Universal Robots URScript: draw_back.script

def unnamed():
  set_tcp(p[0.0,0.0,0.0,0.0,0.0,0.0])
  set_safety_mode_transition_hardness(1)
  set_tool_communication(True, 1000000, 2, 1, 1.5, 3.5)
  set_tool_output_mode(0)
  set_tool_digital_output_mode(0, 1)
  set_tool_digital_output_mode(1, 1)
  set_tool_voltage(0)
  step_count_92a71080_320b_48c3_b710_fb27a0ae3266 = 0.0
  thread Step_Counter_Thread_29a6b4c0_57cd_4359_a365_f92f2370702e():
    while (True):
      step_count_92a71080_320b_48c3_b710_fb27a0ae3266 = step_count_92a71080_320b_48c3_b710_fb27a0ae3266 + 1.0
      sync()
    end
  end
  run Step_Counter_Thread_29a6b4c0_57cd_4359_a365_f92f2370702e()
  set_gravity([0.0, 0.0, 9.82])
  set_standard_analog_input_domain(0, 1)
  set_standard_analog_input_domain(1, 1)
  set_tool_analog_input_domain(0, 1)
  set_tool_analog_input_domain(1, 1)
  set_analog_outputdomain(0, 0)
  set_analog_outputdomain(1, 0)
  set_input_actions_to_default()
  set_target_payload(1.070000, [0.002000, 0.003000, 0.057000], [0.001723, 0.001723, 0.001723, 0.000000, 0.000000, 0.000000])
  global Plane_1=p[-0.700006141123905,1.3454883874109249E-6,0.3910559577028425,-1.2089868272251132,-1.2089999932245832,1.20858562628424]
  global Plane_2=p[0.0,0.0,0.0,0.0,0.0,0.0]
  global Point_1=p[0.6913645118948067,-0.12399382748223003,0.49223711947071,-1.2983729986843258,1.1259514972191385,-1.2203503861141718]
  $ 1 "Robot Program"
  $ 2 "Script: draw_back.script"
  def Machining1():
    # Default parameters:
    global speed_ms = 0.3
    global speed_rads = 0.75
    global accel_mss = 3
    global accel_radss = 1.2
    global blend_radius_m = 0.001

    # Add subprograms here
    # Start of main program
    # Program generated by RoboDK v5.6.5 for UR10e on 18/10/2023 16:38:27
    # Using nominal kinematics.
    blend_radius_m = 0.001
    speed_ms = 1.000
    # set_reference(p[0.335000, -0.152000, 0.000000, 0.000000, 0.000000, 0.000000])
    set_tcp(p[0.000000, 0.000000, 0.252000, 0.000000, 0.000000, 0.000000])
    # Show Tool
    movej([0.136763, -1.127639, -2.609664, -0.975086, 1.570796, 1.707559],accel_radss,speed_rads,0,blend_radius_m)
    movel([0.136763, -1.187625, -2.647719, -0.877045, 1.570796, 1.707559],accel_mss,speed_ms,0,blend_radius_m)
    speed_ms = 1.000
    movel([0.136763, -1.198811, -2.653791, -0.859786, 1.570796, 1.707559],accel_mss,speed_ms,0,blend_radius_m)
    movel([0.136763, -1.222268, -2.665681, -0.824440, 1.570796, 1.707559],accel_mss,speed_ms,0,blend_radius_m)
    movel([0.124896, -1.226310, -2.663645, -0.822433, 1.570796, 1.695693],accel_mss,speed_ms,0,blend_radius_m)
    movel([0.124896, -1.202890, -2.651801, -0.857697, 1.570796, 1.695693],accel_mss,speed_ms,0,blend_radius_m)
    movel([0.135681, -1.206174, -2.650186, -0.856029, 1.570796, 1.706478],accel_mss,speed_ms,0,blend_radius_m)
    movel([0.135681, -1.229564, -2.661993, -0.820832, 1.570796, 1.706478],accel_mss,speed_ms,0,blend_radius_m)
    movel([0.123913, -1.233531, -2.659963, -0.818895, 1.570796, 1.694709],accel_mss,speed_ms,0,blend_radius_m)
    movel([0.123913, -1.210179, -2.648200, -0.854011, 1.570796, 1.694709],accel_mss,speed_ms,0,blend_radius_m)
    movel([0.131108, -1.200743, -2.652851, -0.858795, 1.570796, 1.701904],accel_mss,speed_ms,0,blend_radius_m)
    movel([0.131108, -1.224182, -2.664719, -0.823487, 1.570796, 1.701904],accel_mss,speed_ms,0,blend_radius_m)
    movel([0.130073, -1.231443, -2.661034, -0.819912, 1.570796, 1.700869],accel_mss,speed_ms,0,blend_radius_m)
    movel([0.130073, -1.208071, -2.649247, -0.855071, 1.570796, 1.700869],accel_mss,speed_ms,0,blend_radius_m)
    movel([0.135147, -1.209825, -2.648376, -0.854188, 1.570796, 1.705943],accel_mss,speed_ms,0,blend_radius_m)
    movel([0.135147, -1.233181, -2.660143, -0.819066, 1.570796, 1.705943],accel_mss,speed_ms,0,blend_radius_m)
    movel([0.134512, -1.233881, -2.659782, -0.818725, 1.570796, 1.705309],accel_mss,speed_ms,0,blend_radius_m)
    movel([0.134995, -1.234210, -2.659613, -0.818566, 1.570796, 1.705792],accel_mss,speed_ms,0,blend_radius_m)
    movel([0.135630, -1.233511, -2.659973, -0.818905, 1.570796, 1.706426],accel_mss,speed_ms,0,blend_radius_m)
    movel([0.135147, -1.233181, -2.660143, -0.819066, 1.570796, 1.705943],accel_mss,speed_ms,0,blend_radius_m)
    movel([0.135147, -1.209825, -2.648376, -0.854188, 1.570796, 1.705943],accel_mss,speed_ms,0,blend_radius_m)
    movel([0.131163, -1.211657, -2.647462, -0.853270, 1.570796, 1.701959],accel_mss,speed_ms,0,blend_radius_m)
    movel([0.131163, -1.234995, -2.659208, -0.818185, 1.570796, 1.701959],accel_mss,speed_ms,0,blend_radius_m)
    movel([0.123358, -1.237621, -2.657850, -0.816918, 1.570796, 1.694154],accel_mss,speed_ms,0,blend_radius_m)
    movel([0.123358, -1.214308, -2.646133, -0.851948, 1.570796, 1.694154],accel_mss,speed_ms,0,blend_radius_m)
    movel([0.118731, -1.205544, -2.650497, -0.856348, 1.570796, 1.689527],accel_mss,speed_ms,0,blend_radius_m)
    movel([0.118731, -1.228940, -2.662311, -0.821138, 1.570796, 1.689527],accel_mss,speed_ms,0,blend_radius_m)
    movel([0.109176, -1.232299, -2.660595, -0.819495, 1.570796, 1.679972],accel_mss,speed_ms,0,blend_radius_m)
    movel([0.107432, -1.233406, -2.660027, -0.818956, 1.570796, 1.678228],accel_mss,speed_ms,0,blend_radius_m)
    movel([0.106751, -1.234624, -2.659400, -0.818365, 1.570796, 1.677547],accel_mss,speed_ms,0,blend_radius_m)
    movel([0.106631, -1.235641, -2.658875, -0.817873, 1.570796, 1.677427],accel_mss,speed_ms,0,blend_radius_m)
    movel([0.106631, -1.212309, -2.647136, -0.852944, 1.570796, 1.677427],accel_mss,speed_ms,0,blend_radius_m)
    movel([0.114988, -1.205377, -2.650579, -0.856433, 1.570796, 1.685784],accel_mss,speed_ms,0,blend_radius_m)
    movel([0.114988, -1.228774, -2.662396, -0.821219, 1.570796, 1.685784],accel_mss,speed_ms,0,blend_radius_m)
    movel([0.114535, -1.232368, -2.660560, -0.819461, 1.570796, 1.685331],accel_mss,speed_ms,0,blend_radius_m)
    movel([0.114535, -1.209004, -2.648784, -0.854601, 1.570796, 1.685331],accel_mss,speed_ms,0,blend_radius_m)
    movel([0.117997, -1.211242, -2.647669, -0.853477, 1.570796, 1.688794],accel_mss,speed_ms,0,blend_radius_m)
    movel([0.117997, -1.234584, -2.659420, -0.818384, 1.570796, 1.688794],accel_mss,speed_ms,0,blend_radius_m)
    movel([0.106273, -1.238681, -2.657299, -0.816409, 1.570796, 1.677069],accel_mss,speed_ms,0,blend_radius_m)
    movel([0.106273, -1.215379, -2.645594, -0.851416, 1.570796, 1.677069],accel_mss,speed_ms,0,blend_radius_m)
    movel([0.111851, -1.213399, -2.646590, -0.852400, 1.570796, 1.682647],accel_mss,speed_ms,0,blend_radius_m)
    movel([0.111851, -1.236721, -2.658316, -0.817352, 1.570796, 1.682647],accel_mss,speed_ms,0,blend_radius_m)
    movel([0.113335, -1.237661, -2.657829, -0.816899, 1.570796, 1.684132],accel_mss,speed_ms,0,blend_radius_m)
    movel([0.113766, -1.238482, -2.657402, -0.816505, 1.570796, 1.684562],accel_mss,speed_ms,0,blend_radius_m)
    movel([0.113575, -1.240002, -2.656611, -0.815777, 1.570796, 1.684371],accel_mss,speed_ms,0,blend_radius_m)
    movel([0.112893, -1.241205, -2.655982, -0.815202, 1.570796, 1.683689],accel_mss,speed_ms,0,blend_radius_m)
    movel([0.111165, -1.242286, -2.655416, -0.814687, 1.570796, 1.681962],accel_mss,speed_ms,0,blend_radius_m)
    movel([0.105623, -1.244218, -2.654400, -0.813771, 1.570796, 1.676419],accel_mss,speed_ms,0,blend_radius_m)
    movel([0.105623, -1.220971, -2.642758, -0.848660, 1.570796, 1.676419],accel_mss,speed_ms,0,blend_radius_m)
    movel([0.112197, -1.227862, -2.639215, -0.845312, 1.570796, 1.682993],accel_mss,speed_ms,0,blend_radius_m)
    movel([0.112197, -1.251037, -2.650780, -0.810572, 1.570796, 1.682993],accel_mss,speed_ms,0,blend_radius_m)
    movel([0.104520, -1.253671, -2.649367, -0.809351, 1.570796, 1.675316],accel_mss,speed_ms,0,blend_radius_m)
    movel([0.104520, -1.230524, -2.637832, -0.844033, 1.570796, 1.675316],accel_mss,speed_ms,0,blend_radius_m)
    movel([0.110550, -1.228429, -2.638921, -0.845039, 1.570796, 1.681347],accel_mss,speed_ms,0,blend_radius_m)
    movel([0.110550, -1.251599, -2.650480, -0.810311, 1.570796, 1.681347],accel_mss,speed_ms,0,blend_radius_m)
    movel([0.111771, -1.250229, -2.651212, -0.810948, 1.570796, 1.682568],accel_mss,speed_ms,0,blend_radius_m)
    movel([0.112445, -1.249045, -2.651844, -0.811501, 1.570796, 1.683241],accel_mss,speed_ms,0,blend_radius_m)
    movel([0.112632, -1.247546, -2.652640, -0.812202, 1.570796, 1.683428],accel_mss,speed_ms,0,blend_radius_m)
    movel([0.112205, -1.246735, -2.653071, -0.812584, 1.570796, 1.683001],accel_mss,speed_ms,0,blend_radius_m)
    movel([0.111225, -1.246113, -2.653400, -0.812876, 1.570796, 1.682021],accel_mss,speed_ms,0,blend_radius_m)
    movel([0.109629, -1.246184, -2.653362, -0.812843, 1.570796, 1.680426],accel_mss,speed_ms,0,blend_radius_m)
    movel([0.108525, -1.246566, -2.653160, -0.812663, 1.570796, 1.679321],accel_mss,speed_ms,0,blend_radius_m)
    movel([0.106810, -1.247640, -2.652591, -0.812159, 1.570796, 1.677606],accel_mss,speed_ms,0,blend_radius_m)
    movel([0.105590, -1.249019, -2.651857, -0.811513, 1.570796, 1.676386],accel_mss,speed_ms,0,blend_radius_m)
    movel([0.104923, -1.250204, -2.651225, -0.810959, 1.570796, 1.675720],accel_mss,speed_ms,0,blend_radius_m)
    movel([0.104750, -1.251692, -2.650430, -0.810267, 1.570796, 1.675546],accel_mss,speed_ms,0,blend_radius_m)
    movel([0.105183, -1.252493, -2.650000, -0.809896, 1.570796, 1.675979],accel_mss,speed_ms,0,blend_radius_m)
    movel([0.106163, -1.253104, -2.649672, -0.809613, 1.570796, 1.676960],accel_mss,speed_ms,0,blend_radius_m)
    movel([0.106163, -1.229951, -2.638130, -0.844308, 1.570796, 1.676960],accel_mss,speed_ms,0,blend_radius_m)
    movel([0.111704, -1.231871, -2.637129, -0.843390, 1.570796, 1.682501],accel_mss,speed_ms,0,blend_radius_m)
    movel([0.111704, -1.255003, -2.648649, -0.808736, 1.570796, 1.682501],accel_mss,speed_ms,0,blend_radius_m)
    movel([0.104062, -1.257611, -2.647238, -0.807540, 1.570796, 1.674858],accel_mss,speed_ms,0,blend_radius_m)
    movel([0.104062, -1.234506, -2.635747, -0.842136, 1.570796, 1.674858],accel_mss,speed_ms,0,blend_radius_m)
    movel([0.109519, -1.232620, -2.636737, -0.843032, 1.570796, 1.680315],accel_mss,speed_ms,0,blend_radius_m)
    movel([0.109519, -1.255745, -2.648249, -0.808395, 1.570796, 1.680315],accel_mss,speed_ms,0,blend_radius_m)
    movel([0.110975, -1.256669, -2.647749, -0.807971, 1.570796, 1.681772],accel_mss,speed_ms,0,blend_radius_m)
    movel([0.111399, -1.257470, -2.647314, -0.807605, 1.570796, 1.682195],accel_mss,speed_ms,0,blend_radius_m)
    movel([0.111216, -1.258945, -2.646512, -0.806931, 1.570796, 1.682013],accel_mss,speed_ms,0,blend_radius_m)
    movel([0.110551, -1.260110, -2.645877, -0.806401, 1.570796, 1.681348],accel_mss,speed_ms,0,blend_radius_m)
    movel([0.108863, -1.261149, -2.645310, -0.805930, 1.570796, 1.679659],accel_mss,speed_ms,0,blend_radius_m)
    movel([0.103439, -1.262988, -2.644301, -0.805100, 1.570796, 1.674236],accel_mss,speed_ms,0,blend_radius_m)
    movel([0.103439, -1.239944, -2.632871, -0.839574, 1.570796, 1.674236],accel_mss,speed_ms,0,blend_radius_m)
    movel([0.114338, -1.240023, -2.632829, -0.839537, 1.570796, 1.685135],accel_mss,speed_ms,0,blend_radius_m)
    movel([0.114338, -1.263067, -2.644258, -0.805064, 1.570796, 1.685135],accel_mss,speed_ms,0,blend_radius_m)
    movel([0.102991, -1.266871, -2.642159, -0.803359, 1.570796, 1.673788],accel_mss,speed_ms,0,blend_radius_m)
    movel([0.102991, -1.243871, -2.630773, -0.837745, 1.570796, 1.673788],accel_mss,speed_ms,0,blend_radius_m)
    movel([0.109955, -1.246207, -2.629516, -0.836666, 1.570796, 1.680751],accel_mss,speed_ms,0,blend_radius_m)
    movel([0.109955, -1.269180, -2.640876, -0.802333, 1.570796, 1.680751],accel_mss,speed_ms,0,blend_radius_m)
    movel([0.105150, -1.266141, -2.642563, -0.803685, 1.570796, 1.675946],accel_mss,speed_ms,0,blend_radius_m)
    movel([0.105150, -1.243132, -2.631169, -0.838088, 1.570796, 1.675946],accel_mss,speed_ms,0,blend_radius_m)
    movel([0.107078, -1.244359, -2.630511, -0.837519, 1.570796, 1.677874],accel_mss,speed_ms,0,blend_radius_m)
    movel([0.107078, -1.267353, -2.641891, -0.803144, 1.570796, 1.677874],accel_mss,speed_ms,0,blend_radius_m)
    movel([0.102382, -1.272173, -2.639204, -0.801013, 1.570796, 1.673178],accel_mss,speed_ms,0,blend_radius_m)
    movel([0.102382, -1.249235, -2.627877, -0.835277, 1.570796, 1.673178],accel_mss,speed_ms,0,blend_radius_m)
    movel([0.108723, -1.256402, -2.623955, -0.832032, 1.570796, 1.679519],accel_mss,speed_ms,0,blend_radius_m)
    movel([0.108723, -1.279255, -2.635202, -0.797933, 1.570796, 1.679519],accel_mss,speed_ms,0,blend_radius_m)
    movel([0.100970, -1.284533, -2.632178, -0.795678, 1.570796, 1.671766],accel_mss,speed_ms,0,blend_radius_m)
    movel([0.100970, -1.261746, -2.620991, -0.829652, 1.570796, 1.671766],accel_mss,speed_ms,0,blend_radius_m)
    movel([0.108032, -1.262159, -2.620760, -0.829470, 1.570796, 1.678828],accel_mss,speed_ms,0,blend_radius_m)
    movel([0.108032, -1.284942, -2.631943, -0.795505, 1.570796, 1.678828],accel_mss,speed_ms,0,blend_radius_m)
    movel([0.100970, -1.284533, -2.632178, -0.795678, 1.570796, 1.671766],accel_mss,speed_ms,0,blend_radius_m)
    movel([0.098961, -1.284292, -2.632317, -0.795780, 1.570796, 1.669758],accel_mss,speed_ms,0,blend_radius_m)
    movel([0.098008, -1.283703, -2.632656, -0.796030, 1.570796, 1.668804],accel_mss,speed_ms,0,blend_radius_m)
    movel([0.097582, -1.282937, -2.633096, -0.796356, 1.570796, 1.668379],accel_mss,speed_ms,0,blend_radius_m)
    movel([0.097634, -1.282466, -2.633367, -0.796557, 1.570796, 1.668431],accel_mss,speed_ms,0,blend_radius_m)
    movel([0.097634, -1.259652, -2.622156, -0.830581, 1.570796, 1.668431],accel_mss,speed_ms,0,blend_radius_m)
    movel([0.107462, -1.266919, -2.618088, -0.827381, 1.570796, 1.678259],accel_mss,speed_ms,0,blend_radius_m)
    movel([0.107462, -1.289643, -2.629218, -0.793529, 1.570796, 1.678259],accel_mss,speed_ms,0,blend_radius_m)
    movel([0.107050, -1.288875, -2.629665, -0.793849, 1.570796, 1.677846],accel_mss,speed_ms,0,blend_radius_m)
    movel([0.106111, -1.288277, -2.630012, -0.794100, 1.570796, 1.676908],accel_mss,speed_ms,0,blend_radius_m)
    movel([0.104589, -1.288319, -2.629988, -0.794082, 1.570796, 1.675386],accel_mss,speed_ms,0,blend_radius_m)
    movel([0.103537, -1.288662, -2.629789, -0.793939, 1.570796, 1.674334],accel_mss,speed_ms,0,blend_radius_m)
    movel([0.101907, -1.289644, -2.629217, -0.793528, 1.570796, 1.672703],accel_mss,speed_ms,0,blend_radius_m)
    movel([0.100750, -1.290921, -2.628472, -0.792996, 1.570796, 1.671547],accel_mss,speed_ms,0,blend_radius_m)
    movel([0.100120, -1.292024, -2.627826, -0.792538, 1.570796, 1.670917],accel_mss,speed_ms,0,blend_radius_m)
    movel([0.099963, -1.293419, -2.627008, -0.791962, 1.570796, 1.670759],accel_mss,speed_ms,0,blend_radius_m)
    movel([0.100380, -1.294178, -2.626562, -0.791649, 1.570796, 1.671177],accel_mss,speed_ms,0,blend_radius_m)
    movel([0.101319, -1.294766, -2.626216, -0.791407, 1.570796, 1.672116],accel_mss,speed_ms,0,blend_radius_m)
    movel([0.102832, -1.294723, -2.626241, -0.791425, 1.570796, 1.673628],accel_mss,speed_ms,0,blend_radius_m)
    movel([0.103877, -1.294386, -2.626440, -0.791563, 1.570796, 1.674673],accel_mss,speed_ms,0,blend_radius_m)
    movel([0.105499, -1.293417, -2.627010, -0.791963, 1.570796, 1.676295],accel_mss,speed_ms,0,blend_radius_m)
    movel([0.106656, -1.292149, -2.627754, -0.792487, 1.570796, 1.677453],accel_mss,speed_ms,0,blend_radius_m)
    movel([0.107293, -1.291046, -2.628399, -0.792944, 1.570796, 1.678089],accel_mss,speed_ms,0,blend_radius_m)
    movel([0.107462, -1.289643, -2.629218, -0.793529, 1.570796, 1.678259],accel_mss,speed_ms,0,blend_radius_m)
    movel([0.107462, -1.266919, -2.618088, -0.827381, 1.570796, 1.678259],accel_mss,speed_ms,0,blend_radius_m)
    movel([0.106620, -1.273998, -2.614064, -0.824327, 1.570796, 1.677416],accel_mss,speed_ms,0,blend_radius_m)
    movel([0.106620, -1.296631, -2.625115, -0.790643, 1.570796, 1.677416],accel_mss,speed_ms,0,blend_radius_m)
    movel([0.101416, -1.298298, -2.624127, -0.789964, 1.570796, 1.672213],accel_mss,speed_ms,0,blend_radius_m)
    movel([0.099805, -1.299262, -2.623554, -0.789573, 1.570796, 1.670601],accel_mss,speed_ms,0,blend_radius_m)
    movel([0.099182, -1.300349, -2.622906, -0.789134, 1.570796, 1.669978],accel_mss,speed_ms,0,blend_radius_m)
    movel([0.099027, -1.301727, -2.622084, -0.788579, 1.570796, 1.669824],accel_mss,speed_ms,0,blend_radius_m)
    movel([0.099442, -1.302476, -2.621635, -0.788278, 1.570796, 1.670239],accel_mss,speed_ms,0,blend_radius_m)
    movel([0.100838, -1.303353, -2.621109, -0.787927, 1.570796, 1.671634],accel_mss,speed_ms,0,blend_radius_m)
    movel([0.100838, -1.280809, -2.610134, -0.821446, 1.570796, 1.671634],accel_mss,speed_ms,0,blend_radius_m)
    movel([0.106010, -1.279142, -2.611101, -0.822146, 1.570796, 1.676806],accel_mss,speed_ms,0,blend_radius_m)
    movel([0.106010, -1.301708, -2.622095, -0.788586, 1.570796, 1.676806],accel_mss,speed_ms,0,blend_radius_m)
    movel([0.098771, -1.304015, -2.620711, -0.787663, 1.570796, 1.669567],accel_mss,speed_ms,0,blend_radius_m)
    movel([0.098771, -1.281481, -2.609743, -0.821165, 1.570796, 1.669567],accel_mss,speed_ms,0,blend_radius_m)
    movel([0.107951, -1.291859, -2.603635, -0.816895, 1.570796, 1.678747],accel_mss,speed_ms,0,blend_radius_m)
    movel([0.107951, -1.314254, -2.614488, -0.783648, 1.570796, 1.678747],accel_mss,speed_ms,0,blend_radius_m)
    movel([0.108062, -1.313350, -2.615042, -0.783996, 1.570796, 1.678858],accel_mss,speed_ms,0,blend_radius_m)
    movel([0.107662, -1.312603, -2.615500, -0.784286, 1.570796, 1.678458],accel_mss,speed_ms,0,blend_radius_m)
    movel([0.106184, -1.312625, -2.615487, -0.784277, 1.570796, 1.676980],accel_mss,speed_ms,0,blend_radius_m)
    movel([0.097508, -1.315340, -2.613819, -0.783230, 1.570796, 1.668304],accel_mss,speed_ms,0,blend_radius_m)
    movel([0.097508, -1.292961, -2.602979, -0.816449, 1.570796, 1.668304],accel_mss,speed_ms,0,blend_radius_m)
    movel([0.104812, -1.289315, -2.605145, -0.817929, 1.570796, 1.675609],accel_mss,speed_ms,0,blend_radius_m)
    movel([0.104812, -1.311744, -2.616026, -0.784619, 1.570796, 1.675609],accel_mss,speed_ms,0,blend_radius_m)
    movel([0.104437, -1.314905, -2.614087, -0.783397, 1.570796, 1.675233],accel_mss,speed_ms,0,blend_radius_m)
    movel([0.104437, -1.292520, -2.603242, -0.816627, 1.570796, 1.675233],accel_mss,speed_ms,0,blend_radius_m)
    movel([0.103853, -1.297526, -2.600243, -0.814620, 1.570796, 1.674649],accel_mss,speed_ms,0,blend_radius_m)
    movel([0.103853, -1.319842, -2.611033, -0.781515, 1.570796, 1.674649],accel_mss,speed_ms,0,blend_radius_m)
    movel([0.103451, -1.319103, -2.611492, -0.781794, 1.570796, 1.674248],accel_mss,speed_ms,0,blend_radius_m)
    movel([0.102542, -1.318522, -2.611853, -0.782015, 1.570796, 1.673338],accel_mss,speed_ms,0,blend_radius_m)
    movel([0.101071, -1.318547, -2.611837, -0.782005, 1.570796, 1.671867],accel_mss,speed_ms,0,blend_radius_m)
    movel([0.100055, -1.318864, -2.611641, -0.781885, 1.570796, 1.670852],accel_mss,speed_ms,0,blend_radius_m)
    movel([0.098483, -1.319785, -2.611068, -0.781536, 1.570796, 1.669279],accel_mss,speed_ms,0,blend_radius_m)
    movel([0.097370, -1.320994, -2.610315, -0.781080, 1.570796, 1.668167],accel_mss,speed_ms,0,blend_radius_m)
    movel([0.096766, -1.322042, -2.609661, -0.780686, 1.570796, 1.667562],accel_mss,speed_ms,0,blend_radius_m)
    movel([0.096619, -1.323374, -2.608828, -0.780188, 1.570796, 1.667415],accel_mss,speed_ms,0,blend_radius_m)
    movel([0.097025, -1.324103, -2.608370, -0.779916, 1.570796, 1.667822],accel_mss,speed_ms,0,blend_radius_m)
    movel([0.097935, -1.324676, -2.608011, -0.779703, 1.570796, 1.668732],accel_mss,speed_ms,0,blend_radius_m)
    movel([0.099397, -1.324650, -2.608027, -0.779712, 1.570796, 1.670194],accel_mss,speed_ms,0,blend_radius_m)
    movel([0.100406, -1.324339, -2.608222, -0.779828, 1.570796, 1.671202],accel_mss,speed_ms,0,blend_radius_m)
    movel([0.101970, -1.323429, -2.608793, -0.780167, 1.570796, 1.672767],accel_mss,speed_ms,0,blend_radius_m)
    movel([0.103084, -1.322228, -2.609545, -0.780616, 1.570796, 1.673880],accel_mss,speed_ms,0,blend_radius_m)
    movel([0.103695, -1.321181, -2.610198, -0.781009, 1.570796, 1.674491],accel_mss,speed_ms,0,blend_radius_m)
    movel([0.103853, -1.319842, -2.611033, -0.781515, 1.570796, 1.674649],accel_mss,speed_ms,0,blend_radius_m)
    movel([0.103853, -1.297526, -2.600243, -0.814620, 1.570796, 1.674649],accel_mss,speed_ms,0,blend_radius_m)
    movel([0.103067, -1.304293, -2.596138, -0.811957, 1.570796, 1.673863],accel_mss,speed_ms,0,blend_radius_m)
    movel([0.103067, -1.326513, -2.606854, -0.779022, 1.570796, 1.673863],accel_mss,speed_ms,0,blend_radius_m)
    movel([0.096035, -1.328675, -2.605486, -0.778227, 1.570796, 1.666831],accel_mss,speed_ms,0,blend_radius_m)
    movel([0.096035, -1.306487, -2.594795, -0.811107, 1.570796, 1.666831],accel_mss,speed_ms,0,blend_radius_m)
    movel([0.100052, -1.305230, -2.595566, -0.811594, 1.570796, 1.670848],accel_mss,speed_ms,0,blend_radius_m)
    movel([0.100052, -1.327436, -2.606271, -0.778682, 1.570796, 1.670848],accel_mss,speed_ms,0,blend_radius_m)
    movel([0.101508, -1.327416, -2.606284, -0.778690, 1.570796, 1.672304],accel_mss,speed_ms,0,blend_radius_m)
    movel([0.102409, -1.327992, -2.605919, -0.778478, 1.570796, 1.673205],accel_mss,speed_ms,0,blend_radius_m)
    movel([0.102807, -1.328722, -2.605457, -0.778210, 1.570796, 1.673604],accel_mss,speed_ms,0,blend_radius_m)
    movel([0.102652, -1.330044, -2.604618, -0.777727, 1.570796, 1.673449],accel_mss,speed_ms,0,blend_radius_m)
    movel([0.102652, -1.307875, -2.593942, -0.810572, 1.570796, 1.673449],accel_mss,speed_ms,0,blend_radius_m)
    movel([0.101682, -1.316308, -2.588706, -0.807375, 1.570796, 1.672478],accel_mss,speed_ms,0,blend_radius_m)
    movel([0.101682, -1.338353, -2.599289, -0.774747, 1.570796, 1.672478],accel_mss,speed_ms,0,blend_radius_m)
    movel([0.094466, -1.343037, -2.596244, -0.773108, 1.570796, 1.665263],accel_mss,speed_ms,0,blend_radius_m)
    movel([0.094466, -1.321062, -2.585713, -0.805613, 1.570796, 1.665263],accel_mss,speed_ms,0,blend_radius_m)
    movel([0.101079, -1.321581, -2.585385, -0.805423, 1.570796, 1.671875],accel_mss,speed_ms,0,blend_radius_m)
    movel([0.101079, -1.343547, -2.595911, -0.772931, 1.570796, 1.671875],accel_mss,speed_ms,0,blend_radius_m)
    movel([0.094466, -1.343037, -2.596244, -0.773108, 1.570796, 1.665263],accel_mss,speed_ms,0,blend_radius_m)
    movel([0.094466, -1.321062, -2.585713, -0.805613, 1.570796, 1.665263],accel_mss,speed_ms,0,blend_radius_m)
    movel([0.104271, -1.322733, -2.584655, -0.805001, 1.570796, 1.675068],accel_mss,speed_ms,0,blend_radius_m)
    movel([0.104271, -1.344682, -2.595168, -0.772539, 1.570796, 1.675068],accel_mss,speed_ms,0,blend_radius_m)
    movel([0.103728, -1.345257, -2.594790, -0.772341, 1.570796, 1.674524],accel_mss,speed_ms,0,blend_radius_m)
    movel([0.104168, -1.345543, -2.594603, -0.772243, 1.570796, 1.674965],accel_mss,speed_ms,0,blend_radius_m)
    movel([0.104711, -1.344968, -2.594980, -0.772441, 1.570796, 1.675508],accel_mss,speed_ms,0,blend_radius_m)
    movel([0.104271, -1.344682, -2.595168, -0.772539, 1.570796, 1.675068],accel_mss,speed_ms,0,blend_radius_m)
    movel([0.104271, -1.322733, -2.584655, -0.805001, 1.570796, 1.675068],accel_mss,speed_ms,0,blend_radius_m)
    movel([0.100780, -1.324202, -2.583721, -0.804466, 1.570796, 1.671576],accel_mss,speed_ms,0,blend_radius_m)
    movel([0.100780, -1.346129, -2.594218, -0.772043, 1.570796, 1.671576],accel_mss,speed_ms,0,blend_radius_m)
    movel([0.093909, -1.348182, -2.592864, -0.771342, 1.570796, 1.664705],accel_mss,speed_ms,0,blend_radius_m)
    movel([0.093909, -1.326287, -2.582390, -0.803712, 1.570796, 1.664705],accel_mss,speed_ms,0,blend_radius_m)
    movel([0.098434, -1.332441, -2.578430, -0.801518, 1.570796, 1.669230],accel_mss,speed_ms,0,blend_radius_m)
    movel([0.098434, -1.354242, -2.588837, -0.769310, 1.570796, 1.669230],accel_mss,speed_ms,0,blend_radius_m)
    movel([0.099455, -1.353532, -2.589312, -0.769545, 1.570796, 1.670252],accel_mss,speed_ms,0,blend_radius_m)
    movel([0.100089, -1.352113, -2.590258, -0.770018, 1.570796, 1.670885],accel_mss,speed_ms,0,blend_radius_m)
    movel([0.100236, -1.350835, -2.591107, -0.770446, 1.570796, 1.671033],accel_mss,speed_ms,0,blend_radius_m)
    movel([0.099895, -1.349700, -2.591861, -0.770829, 1.570796, 1.670691],accel_mss,speed_ms,0,blend_radius_m)
    movel([0.098965, -1.349562, -2.591952, -0.770875, 1.570796, 1.669761],accel_mss,speed_ms,0,blend_radius_m)
    movel([0.097938, -1.350279, -2.591477, -0.770633, 1.570796, 1.668735],accel_mss,speed_ms,0,blend_radius_m)
    movel([0.097354, -1.351276, -2.590815, -0.770298, 1.570796, 1.668151],accel_mss,speed_ms,0,blend_radius_m)
    movel([0.096629, -1.353545, -2.589303, -0.769541, 1.570796, 1.667426],accel_mss,speed_ms,0,blend_radius_m)
    movel([0.096048, -1.354537, -2.588640, -0.769212, 1.570796, 1.666845],accel_mss,speed_ms,0,blend_radius_m)
    movel([0.095029, -1.355248, -2.588163, -0.768977, 1.570796, 1.665825],accel_mss,speed_ms,0,blend_radius_m)
    movel([0.094543, -1.355392, -2.588067, -0.768930, 1.570796, 1.665339],accel_mss,speed_ms,0,blend_radius_m)
    movel([0.093617, -1.355259, -2.588156, -0.768974, 1.570796, 1.664413],accel_mss,speed_ms,0,blend_radius_m)
    movel([0.093267, -1.354135, -2.588909, -0.769345, 1.570796, 1.664063],accel_mss,speed_ms,0,blend_radius_m)
    movel([0.093404, -1.352864, -2.589757, -0.769768, 1.570796, 1.664200],accel_mss,speed_ms,0,blend_radius_m)
    movel([0.094029, -1.351444, -2.590703, -0.770242, 1.570796, 1.664826],accel_mss,speed_ms,0,blend_radius_m)
    movel([0.095053, -1.350726, -2.591180, -0.770483, 1.570796, 1.665849],accel_mss,speed_ms,0,blend_radius_m)
    movel([0.095053, -1.328870, -2.580734, -0.802785, 1.570796, 1.665849],accel_mss,speed_ms,0,blend_radius_m)
    movel([0.103000, -1.333582, -2.577690, -0.801117, 1.570796, 1.673797],accel_mss,speed_ms,0,blend_radius_m)
    movel([0.103000, -1.355366, -2.588084, -0.768939, 1.570796, 1.673797],accel_mss,speed_ms,0,blend_radius_m)
    movel([0.102465, -1.355931, -2.587706, -0.768753, 1.570796, 1.673261],accel_mss,speed_ms,0,blend_radius_m)
    movel([0.102900, -1.356213, -2.587516, -0.768660, 1.570796, 1.673696],accel_mss,speed_ms,0,blend_radius_m)
    movel([0.103436, -1.355649, -2.587895, -0.768845, 1.570796, 1.674232],accel_mss,speed_ms,0,blend_radius_m)
    movel([0.103000, -1.355366, -2.588084, -0.768939, 1.570796, 1.673797],accel_mss,speed_ms,0,blend_radius_m)
    movel([0.103000, -1.333582, -2.577690, -0.801117, 1.570796, 1.673797],accel_mss,speed_ms,0,blend_radius_m)
    movel([0.099553, -1.335016, -2.576758, -0.800615, 1.570796, 1.670350],accel_mss,speed_ms,0,blend_radius_m)
    movel([0.099553, -1.356778, -2.587137, -0.768475, 1.570796, 1.670350],accel_mss,speed_ms,0,blend_radius_m)
    movel([0.092768, -1.358775, -2.585791, -0.767823, 1.570796, 1.663565],accel_mss,speed_ms,0,blend_radius_m)
    movel([0.092768, -1.337045, -2.575434, -0.799910, 1.570796, 1.663565],accel_mss,speed_ms,0,blend_radius_m)
    movel([0.102501, -1.337875, -2.574891, -0.799623, 1.570796, 1.673297],accel_mss,speed_ms,0,blend_radius_m)
    movel([0.102501, -1.359591, -2.585239, -0.767558, 1.570796, 1.673297],accel_mss,speed_ms,0,blend_radius_m)
    movel([0.094293, -1.361979, -2.583620, -0.766789, 1.570796, 1.665090],accel_mss,speed_ms,0,blend_radius_m)
    movel([0.092802, -1.362823, -2.583047, -0.766519, 1.570796, 1.663598],accel_mss,speed_ms,0,blend_radius_m)
    movel([0.092231, -1.363800, -2.582381, -0.766208, 1.570796, 1.663027],accel_mss,speed_ms,0,blend_radius_m)
    movel([0.092142, -1.364634, -2.581811, -0.765944, 1.570796, 1.662938],accel_mss,speed_ms,0,blend_radius_m)
    movel([0.092142, -1.342997, -2.571519, -0.797873, 1.570796, 1.662938],accel_mss,speed_ms,0,blend_radius_m)
    movel([0.099263, -1.337587, -2.575080, -0.799722, 1.570796, 1.670060],accel_mss,speed_ms,0,blend_radius_m)
    movel([0.099263, -1.359308, -2.585431, -0.767650, 1.570796, 1.670060],accel_mss,speed_ms,0,blend_radius_m)
    movel([0.098928, -1.362248, -2.583438, -0.766703, 1.570796, 1.669724],accel_mss,speed_ms,0,blend_radius_m)
    movel([0.098928, -1.340573, -2.573119, -0.798696, 1.570796, 1.669724],accel_mss,speed_ms,0,blend_radius_m)
    movel([0.102006, -1.342140, -2.572086, -0.798163, 1.570796, 1.672802],accel_mss,speed_ms,0,blend_radius_m)
    movel([0.102006, -1.363790, -2.582387, -0.766211, 1.570796, 1.672802],accel_mss,speed_ms,0,blend_radius_m)
    movel([0.101476, -1.364346, -2.582008, -0.766035, 1.570796, 1.672273],accel_mss,speed_ms,0,blend_radius_m)
    movel([0.101908, -1.364627, -2.581816, -0.765946, 1.570796, 1.672704],accel_mss,speed_ms,0,blend_radius_m)
    movel([0.102438, -1.364071, -2.582196, -0.766122, 1.570796, 1.673234],accel_mss,speed_ms,0,blend_radius_m)
    movel([0.102006, -1.363790, -2.582387, -0.766211, 1.570796, 1.672802],accel_mss,speed_ms,0,blend_radius_m)
    movel([0.102006, -1.342140, -2.572086, -0.798163, 1.570796, 1.672802],accel_mss,speed_ms,0,blend_radius_m)
    movel([0.098594, -1.343547, -2.571155, -0.797687, 1.570796, 1.669390],accel_mss,speed_ms,0,blend_radius_m)
    movel([0.098594, -1.365175, -2.581441, -0.765773, 1.570796, 1.669390],accel_mss,speed_ms,0,blend_radius_m)
    movel([0.091876, -1.367129, -2.580102, -0.765158, 1.570796, 1.662673],accel_mss,speed_ms,0,blend_radius_m)
    movel([0.091876, -1.345533, -2.569837, -0.797019, 1.570796, 1.662673],accel_mss,speed_ms,0,blend_radius_m)
    movel([0.098215, -1.346930, -2.568906, -0.796553, 1.570796, 1.669012],accel_mss,speed_ms,0,blend_radius_m)
    movel([0.098215, -1.368504, -2.579156, -0.764729, 1.570796, 1.669012],accel_mss,speed_ms,0,blend_radius_m)
    movel([0.091524, -1.370441, -2.577819, -0.764129, 1.570796, 1.662321],accel_mss,speed_ms,0,blend_radius_m)
    movel([0.091524, -1.348899, -2.567590, -0.795900, 1.570796, 1.662321],accel_mss,speed_ms,0,blend_radius_m)
    movel([0.096302, -1.347490, -2.568533, -0.796367, 1.570796, 1.667099],accel_mss,speed_ms,0,blend_radius_m)
    movel([0.096302, -1.369055, -2.578776, -0.764558, 1.570796, 1.667099],accel_mss,speed_ms,0,blend_radius_m)
    movel([0.097596, -1.369886, -2.578203, -0.764300, 1.570796, 1.668393],accel_mss,speed_ms,0,blend_radius_m)
    movel([0.097980, -1.370577, -2.577725, -0.764087, 1.570796, 1.668777],accel_mss,speed_ms,0,blend_radius_m)
    movel([0.097840, -1.371817, -2.576866, -0.763706, 1.570796, 1.668636],accel_mss,speed_ms,0,blend_radius_m)
    movel([0.097270, -1.372779, -2.576198, -0.763412, 1.570796, 1.668067],accel_mss,speed_ms,0,blend_radius_m)
    movel([0.095797, -1.373599, -2.575628, -0.763162, 1.570796, 1.666593],accel_mss,speed_ms,0,blend_radius_m)
    movel([0.091045, -1.374969, -2.574673, -0.762747, 1.570796, 1.661841],accel_mss,speed_ms,0,blend_radius_m)
    movel([0.091045, -1.353501, -2.564494, -0.794394, 1.570796, 1.661841],accel_mss,speed_ms,0,blend_radius_m)
    movel([0.096822, -1.359472, -2.560433, -0.792484, 1.570796, 1.667618],accel_mss,speed_ms,0,blend_radius_m)
    movel([0.096822, -1.380843, -2.570548, -0.760998, 1.570796, 1.667618],accel_mss,speed_ms,0,blend_radius_m)
    movel([0.089288, -1.382989, -2.569029, -0.760371, 1.570796, 1.660084],accel_mss,speed_ms,0,blend_radius_m)
    movel([0.087918, -1.382990, -2.569028, -0.760371, 1.570796, 1.658714],accel_mss,speed_ms,0,blend_radius_m)
    movel([0.087489, -1.382721, -2.569219, -0.760449, 1.570796, 1.658285],accel_mss,speed_ms,0,blend_radius_m)
    movel([0.087100, -1.382047, -2.569697, -0.760646, 1.570796, 1.657896],accel_mss,speed_ms,0,blend_radius_m)
    movel([0.087224, -1.380829, -2.570558, -0.761002, 1.570796, 1.658020],accel_mss,speed_ms,0,blend_radius_m)
    movel([0.087779, -1.379879, -2.571228, -0.761282, 1.570796, 1.658575],accel_mss,speed_ms,0,blend_radius_m)
    movel([0.087779, -1.358491, -2.561103, -0.792794, 1.570796, 1.658575],accel_mss,speed_ms,0,blend_radius_m)
    movel([0.095408, -1.359878, -2.560155, -0.792356, 1.570796, 1.666204],accel_mss,speed_ms,0,blend_radius_m)
    movel([0.095408, -1.381243, -2.570266, -0.760881, 1.570796, 1.666204],accel_mss,speed_ms,0,blend_radius_m)
    movel([0.096442, -1.380161, -2.571029, -0.761198, 1.570796, 1.667238],accel_mss,speed_ms,0,blend_radius_m)
    movel([0.097005, -1.379211, -2.571699, -0.761479, 1.570796, 1.667802],accel_mss,speed_ms,0,blend_radius_m)
    movel([0.097143, -1.377984, -2.572562, -0.761843, 1.570796, 1.667940],accel_mss,speed_ms,0,blend_radius_m)
    movel([0.096762, -1.377300, -2.573042, -0.762047, 1.570796, 1.667558],accel_mss,speed_ms,0,blend_radius_m)
    movel([0.095907, -1.376750, -2.573428, -0.762212, 1.570796, 1.666703],accel_mss,speed_ms,0,blend_radius_m)
    movel([0.094531, -1.376746, -2.573430, -0.762213, 1.570796, 1.665327],accel_mss,speed_ms,0,blend_radius_m)
    movel([0.093583, -1.377017, -2.573240, -0.762131, 1.570796, 1.664379],accel_mss,speed_ms,0,blend_radius_m)
    movel([0.092119, -1.377834, -2.572667, -0.761888, 1.570796, 1.662915],accel_mss,speed_ms,0,blend_radius_m)
    movel([0.091086, -1.378923, -2.571902, -0.761564, 1.570796, 1.661882],accel_mss,speed_ms,0,blend_radius_m)
    movel([0.090527, -1.379874, -2.571232, -0.761283, 1.570796, 1.661324],accel_mss,speed_ms,0,blend_radius_m)
    movel([0.090399, -1.381095, -2.570370, -0.760924, 1.570796, 1.661195],accel_mss,speed_ms,0,blend_radius_m)
    movel([0.090785, -1.381772, -2.569891, -0.760726, 1.570796, 1.661581],accel_mss,speed_ms,0,blend_radius_m)
    movel([0.091640, -1.382315, -2.569507, -0.760567, 1.570796, 1.662437],accel_mss,speed_ms,0,blend_radius_m)
    movel([0.091640, -1.360967, -2.559408, -0.792013, 1.570796, 1.662437],accel_mss,speed_ms,0,blend_radius_m)
    movel([0.098767, -1.370469, -2.552826, -0.789094, 1.570796, 1.669564],accel_mss,speed_ms,0,blend_radius_m)
    movel([0.098767, -1.391659, -2.562823, -0.757907, 1.570796, 1.669564],accel_mss,speed_ms,0,blend_radius_m)
    movel([0.089343, -1.391181, -2.563168, -0.758040, 1.570796, 1.660140],accel_mss,speed_ms,0,blend_radius_m)
    movel([0.089343, -1.369983, -2.553165, -0.789240, 1.570796, 1.660140],accel_mss,speed_ms,0,blend_radius_m)
    movel([0.098767, -1.370469, -2.552826, -0.789094, 1.570796, 1.669564],accel_mss,speed_ms,0,blend_radius_m)
    movel([0.098767, -1.391659, -2.562823, -0.757907, 1.570796, 1.669564],accel_mss,speed_ms,0,blend_radius_m)
    movel([0.088681, -1.397559, -2.558537, -0.756293, 1.570796, 1.659477],accel_mss,speed_ms,0,blend_radius_m)
    movel([0.088681, -1.376469, -2.548604, -0.787315, 1.570796, 1.659477],accel_mss,speed_ms,0,blend_radius_m)
    movel([0.092476, -1.370271, -2.552965, -0.789154, 1.570796, 1.663272],accel_mss,speed_ms,0,blend_radius_m)
    movel([0.092476, -1.391464, -2.562964, -0.757961, 1.570796, 1.663272],accel_mss,speed_ms,0,blend_radius_m)
    movel([0.092046, -1.395460, -2.560068, -0.756861, 1.570796, 1.662842],accel_mss,speed_ms,0,blend_radius_m)
    movel([0.092046, -1.374334, -2.550112, -0.787943, 1.570796, 1.662842],accel_mss,speed_ms,0,blend_radius_m)
    movel([0.098172, -1.375756, -2.549109, -0.787524, 1.570796, 1.668968],accel_mss,speed_ms,0,blend_radius_m)
    movel([0.098172, -1.396857, -2.559050, -0.756482, 1.570796, 1.668968],accel_mss,speed_ms,0,blend_radius_m)
    movel([0.088476, -1.399540, -2.557087, -0.755762, 1.570796, 1.659272],accel_mss,speed_ms,0,blend_radius_m)
    movel([0.088476, -1.378484, -2.547176, -0.786729, 1.570796, 1.659272],accel_mss,speed_ms,0,blend_radius_m)
    movel([0.097809, -1.378989, -2.546816, -0.786583, 1.570796, 1.668605],accel_mss,speed_ms,0,blend_radius_m)
    movel([0.097809, -1.400036, -2.556723, -0.755630, 1.570796, 1.668605],accel_mss,speed_ms,0,blend_radius_m)
    movel([0.088150, -1.402697, -2.554764, -0.754928, 1.570796, 1.658946],accel_mss,speed_ms,0,blend_radius_m)
    movel([0.088150, -1.381696, -2.544886, -0.785807, 1.570796, 1.658946],accel_mss,speed_ms,0,blend_radius_m)
    movel([0.097809, -1.378989, -2.546816, -0.786583, 1.570796, 1.668605],accel_mss,speed_ms,0,blend_radius_m)
    movel([0.097809, -1.400036, -2.556723, -0.755630, 1.570796, 1.668605],accel_mss,speed_ms,0,blend_radius_m)
    movel([0.097404, -1.403595, -2.554100, -0.754694, 1.570796, 1.668200],accel_mss,speed_ms,0,blend_radius_m)
    movel([0.096812, -1.404901, -2.553133, -0.754355, 1.570796, 1.667608],accel_mss,speed_ms,0,blend_radius_m)
    movel([0.096310, -1.405418, -2.552749, -0.754221, 1.570796, 1.667106],accel_mss,speed_ms,0,blend_radius_m)
    movel([0.095351, -1.406059, -2.552273, -0.754056, 1.570796, 1.666147],accel_mss,speed_ms,0,blend_radius_m)
    movel([0.094437, -1.406308, -2.552089, -0.753993, 1.570796, 1.665233],accel_mss,speed_ms,0,blend_radius_m)
    movel([0.093565, -1.406164, -2.552195, -0.754029, 1.570796, 1.664362],accel_mss,speed_ms,0,blend_radius_m)
    movel([0.093151, -1.405897, -2.552394, -0.754098, 1.570796, 1.663947],accel_mss,speed_ms,0,blend_radius_m)
    movel([0.092821, -1.404843, -2.553176, -0.754370, 1.570796, 1.663617],accel_mss,speed_ms,0,blend_radius_m)
    movel([0.093206, -1.401296, -2.555797, -0.755296, 1.570796, 1.664003],accel_mss,speed_ms,0,blend_radius_m)
    movel([0.093206, -1.380270, -2.545904, -0.786215, 1.570796, 1.664003],accel_mss,speed_ms,0,blend_radius_m)
    movel([0.092906, -1.383079, -2.543896, -0.785414, 1.570796, 1.663703],accel_mss,speed_ms,0,blend_radius_m)
    movel([0.092906, -1.404056, -2.553759, -0.754574, 1.570796, 1.663703],accel_mss,speed_ms,0,blend_radius_m)
    movel([0.087585, -1.408187, -2.550689, -0.753513, 1.570796, 1.658381],accel_mss,speed_ms,0,blend_radius_m)
    movel([0.087585, -1.387281, -2.540870, -0.784238, 1.570796, 1.658381],accel_mss,speed_ms,0,blend_radius_m)
    movel([0.096166, -1.393755, -2.536160, -0.782474, 1.570796, 1.666962],accel_mss,speed_ms,0,blend_radius_m)
    movel([0.096166, -1.414550, -2.545910, -0.751929, 1.570796, 1.666962],accel_mss,speed_ms,0,blend_radius_m)
    movel([0.086673, -1.417112, -2.543969, -0.751308, 1.570796, 1.657469],accel_mss,speed_ms,0,blend_radius_m)
    movel([0.086205, -1.421723, -2.540451, -0.750215, 1.570796, 1.657001],accel_mss,speed_ms,0,blend_radius_m)
    movel([0.086205, -1.401056, -2.530777, -0.780557, 1.570796, 1.657001],accel_mss,speed_ms,0,blend_radius_m)
    movel([0.095215, -1.402392, -2.529783, -0.780214, 1.570796, 1.666011],accel_mss,speed_ms,0,blend_radius_m)
    movel([0.095215, -1.423036, -2.539444, -0.749910, 1.570796, 1.666011],accel_mss,speed_ms,0,blend_radius_m)
    movel([0.086127, -1.422489, -2.539864, -0.750037, 1.570796, 1.656923],accel_mss,speed_ms,0,blend_radius_m)
    movel([0.086127, -1.401835, -2.530198, -0.780356, 1.570796, 1.656923],accel_mss,speed_ms,0,blend_radius_m)
    movel([0.095215, -1.402392, -2.529783, -0.780214, 1.570796, 1.666011],accel_mss,speed_ms,0,blend_radius_m)
    movel([0.095215, -1.423036, -2.539444, -0.749910, 1.570796, 1.666011],accel_mss,speed_ms,0,blend_radius_m)
    movel([0.085512, -1.428583, -2.535158, -0.748648, 1.570796, 1.656308],accel_mss,speed_ms,0,blend_radius_m)
    movel([0.085512, -1.408038, -2.525556, -0.778794, 1.570796, 1.656308],accel_mss,speed_ms,0,blend_radius_m)
    movel([0.089148, -1.402141, -2.529970, -0.780278, 1.570796, 1.659944],accel_mss,speed_ms,0,blend_radius_m)
    movel([0.089148, -1.422790, -2.539633, -0.749967, 1.570796, 1.659944],accel_mss,speed_ms,0,blend_radius_m)
    movel([0.088749, -1.426607, -2.536690, -0.749092, 1.570796, 1.659546],accel_mss,speed_ms,0,blend_radius_m)
    movel([0.088749, -1.406026, -2.527068, -0.779295, 1.570796, 1.659546],accel_mss,speed_ms,0,blend_radius_m)
    movel([0.094662, -1.407446, -2.526002, -0.778941, 1.570796, 1.665458],accel_mss,speed_ms,0,blend_radius_m)
    movel([0.094662, -1.428002, -2.535609, -0.748778, 1.570796, 1.665458],accel_mss,speed_ms,0,blend_radius_m)
    movel([0.085321, -1.430477, -2.533684, -0.748228, 1.570796, 1.656118],accel_mss,speed_ms,0,blend_radius_m)
    movel([0.085321, -1.409966, -2.524103, -0.778320, 1.570796, 1.656118],accel_mss,speed_ms,0,blend_radius_m)
    movel([0.094662, -1.407446, -2.526002, -0.778941, 1.570796, 1.665458],accel_mss,speed_ms,0,blend_radius_m)
    movel([0.094662, -1.428002, -2.535609, -0.748778, 1.570796, 1.665458],accel_mss,speed_ms,0,blend_radius_m)
    movel([0.094283, -1.431419, -2.532949, -0.748021, 1.570796, 1.665079],accel_mss,speed_ms,0,blend_radius_m)
    movel([0.093715, -1.432669, -2.531971, -0.747748, 1.570796, 1.664511],accel_mss,speed_ms,0,blend_radius_m)
    movel([0.093231, -1.433163, -2.531585, -0.747641, 1.570796, 1.664027],accel_mss,speed_ms,0,blend_radius_m)
    movel([0.092305, -1.433771, -2.531108, -0.747510, 1.570796, 1.663101],accel_mss,speed_ms,0,blend_radius_m)
    movel([0.091420, -1.434002, -2.530927, -0.747460, 1.570796, 1.662217],accel_mss,speed_ms,0,blend_radius_m)
    movel([0.090576, -1.433857, -2.531041, -0.747491, 1.570796, 1.661372],accel_mss,speed_ms,0,blend_radius_m)
    movel([0.090174, -1.433596, -2.531246, -0.747548, 1.570796, 1.660970],accel_mss,speed_ms,0,blend_radius_m)
    movel([0.089851, -1.432580, -2.532041, -0.747768, 1.570796, 1.660647],accel_mss,speed_ms,0,blend_radius_m)
    movel([0.089851, -1.412107, -2.522482, -0.777800, 1.570796, 1.660647],accel_mss,speed_ms,0,blend_radius_m)
    movel([0.090212, -1.408639, -2.525104, -0.778646, 1.570796, 1.661008],accel_mss,speed_ms,0,blend_radius_m)
    movel([0.090212, -1.429173, -2.534699, -0.748516, 1.570796, 1.661008],accel_mss,speed_ms,0,blend_radius_m)
    movel([0.089851, -1.432580, -2.532041, -0.747768, 1.570796, 1.660647],accel_mss,speed_ms,0,blend_radius_m)
    movel([0.089289, -1.433829, -2.531063, -0.747497, 1.570796, 1.660085],accel_mss,speed_ms,0,blend_radius_m)
    movel([0.088807, -1.434322, -2.530676, -0.747391, 1.570796, 1.659604],accel_mss,speed_ms,0,blend_radius_m)
    movel([0.087884, -1.434932, -2.530197, -0.747261, 1.570796, 1.658681],accel_mss,speed_ms,0,blend_radius_m)
    movel([0.086559, -1.435282, -2.529921, -0.747186, 1.570796, 1.657355],accel_mss,speed_ms,0,blend_radius_m)
    movel([0.085714, -1.435141, -2.530032, -0.747216, 1.570796, 1.656510],accel_mss,speed_ms,0,blend_radius_m)
    movel([0.085310, -1.434883, -2.530235, -0.747271, 1.570796, 1.656106],accel_mss,speed_ms,0,blend_radius_m)
    movel([0.084981, -1.433872, -2.531028, -0.747488, 1.570796, 1.655777],accel_mss,speed_ms,0,blend_radius_m)
    movel([0.085321, -1.430477, -2.533684, -0.748228, 1.570796, 1.656118],accel_mss,speed_ms,0,blend_radius_m)
    movel([0.085321, -1.409966, -2.524103, -0.778320, 1.570796, 1.656118],accel_mss,speed_ms,0,blend_radius_m)
    movel([0.096789, -1.214889, -2.645841, -0.851659, 1.570796, 1.667586],accel_mss,speed_ms,0,blend_radius_m)
    movel([0.096789, -1.238196, -2.657551, -0.816642, 1.570796, 1.667586],accel_mss,speed_ms,0,blend_radius_m)
    movel([0.096339, -1.237390, -2.657970, -0.817030, 1.570796, 1.667135],accel_mss,speed_ms,0,blend_radius_m)
    movel([0.095329, -1.236787, -2.658282, -0.817320, 1.570796, 1.666125],accel_mss,speed_ms,0,blend_radius_m)
    movel([0.093704, -1.236893, -2.658227, -0.817269, 1.570796, 1.664501],accel_mss,speed_ms,0,blend_radius_m)
    movel([0.092586, -1.237302, -2.658015, -0.817072, 1.570796, 1.663382],accel_mss,speed_ms,0,blend_radius_m)
    movel([0.090859, -1.238420, -2.657435, -0.816535, 1.570796, 1.661655],accel_mss,speed_ms,0,blend_radius_m)
    movel([0.089642, -1.239833, -2.656699, -0.815857, 1.570796, 1.660438],accel_mss,speed_ms,0,blend_radius_m)
    movel([0.088985, -1.241039, -2.656069, -0.815281, 1.570796, 1.659781],accel_mss,speed_ms,0,blend_radius_m)
    movel([0.088836, -1.242538, -2.655283, -0.814568, 1.570796, 1.659632],accel_mss,speed_ms,0,blend_radius_m)
    movel([0.089293, -1.243333, -2.654866, -0.814190, 1.570796, 1.660089],accel_mss,speed_ms,0,blend_radius_m)
    movel([0.090302, -1.243925, -2.654554, -0.813909, 1.570796, 1.661099],accel_mss,speed_ms,0,blend_radius_m)
    movel([0.091916, -1.243819, -2.654610, -0.813960, 1.570796, 1.662712],accel_mss,speed_ms,0,blend_radius_m)
    movel([0.093026, -1.243417, -2.654822, -0.814150, 1.570796, 1.663822],accel_mss,speed_ms,0,blend_radius_m)
    movel([0.094744, -1.242315, -2.655400, -0.814673, 1.570796, 1.665541],accel_mss,speed_ms,0,blend_radius_m)
    movel([0.095963, -1.240912, -2.656135, -0.815342, 1.570796, 1.666759],accel_mss,speed_ms,0,blend_radius_m)
    movel([0.096627, -1.239706, -2.656765, -0.815918, 1.570796, 1.667423],accel_mss,speed_ms,0,blend_radius_m)
    movel([0.096789, -1.238196, -2.657551, -0.816642, 1.570796, 1.667586],accel_mss,speed_ms,0,blend_radius_m)
    movel([0.096789, -1.214889, -2.645841, -0.851659, 1.570796, 1.667586],accel_mss,speed_ms,0,blend_radius_m)
    movel([0.095983, -1.222481, -2.641987, -0.847922, 1.570796, 1.666780],accel_mss,speed_ms,0,blend_radius_m)
    movel([0.095983, -1.245712, -2.653612, -0.813065, 1.570796, 1.666780],accel_mss,speed_ms,0,blend_radius_m)
    movel([0.088246, -1.248500, -2.652134, -0.811755, 1.570796, 1.659042],accel_mss,speed_ms,0,blend_radius_m)
    movel([0.088246, -1.225298, -2.640540, -0.846551, 1.570796, 1.659042],accel_mss,speed_ms,0,blend_radius_m)
    movel([0.093771, -1.223282, -2.641576, -0.847531, 1.570796, 1.664567],accel_mss,speed_ms,0,blend_radius_m)
    movel([0.093771, -1.246505, -2.653192, -0.812692, 1.570796, 1.664567],accel_mss,speed_ms,0,blend_radius_m)
    movel([0.095271, -1.247402, -2.652717, -0.812270, 1.570796, 1.666068],accel_mss,speed_ms,0,blend_radius_m)
    movel([0.095718, -1.248198, -2.652294, -0.811897, 1.570796, 1.666514],accel_mss,speed_ms,0,blend_radius_m)
    movel([0.095559, -1.249685, -2.651502, -0.811201, 1.570796, 1.666355],accel_mss,speed_ms,0,blend_radius_m)
    movel([0.094903, -1.250871, -2.650869, -0.810649, 1.570796, 1.665700],accel_mss,speed_ms,0,blend_radius_m)
    movel([0.093202, -1.251951, -2.650291, -0.810147, 1.570796, 1.663998],accel_mss,speed_ms,0,blend_radius_m)
    movel([0.087712, -1.253918, -2.649234, -0.809237, 1.570796, 1.658509],accel_mss,speed_ms,0,blend_radius_m)
    movel([0.087712, -1.230773, -2.637702, -0.843914, 1.570796, 1.658509],accel_mss,speed_ms,0,blend_radius_m)
    movel([0.097954, -1.238537, -2.633618, -0.840233, 1.570796, 1.668751],accel_mss,speed_ms,0,blend_radius_m)
    movel([0.097954, -1.261597, -2.645064, -0.805727, 1.570796, 1.668751],accel_mss,speed_ms,0,blend_radius_m)
    movel([0.086570, -1.265585, -2.642871, -0.803934, 1.570796, 1.657366],accel_mss,speed_ms,0,blend_radius_m)
    movel([0.086570, -1.242570, -2.631470, -0.838349, 1.570796, 1.657366],accel_mss,speed_ms,0,blend_radius_m)
    movel([0.097954, -1.238537, -2.633618, -0.840233, 1.570796, 1.668751],accel_mss,speed_ms,0,blend_radius_m)
    movel([0.097954, -1.261597, -2.645064, -0.805727, 1.570796, 1.668751],accel_mss,speed_ms,0,blend_radius_m)
    movel([0.097476, -1.265964, -2.642661, -0.803764, 1.570796, 1.668273],accel_mss,speed_ms,0,blend_radius_m)
    movel([0.096779, -1.267599, -2.641755, -0.803035, 1.570796, 1.667575],accel_mss,speed_ms,0,blend_radius_m)
    movel([0.096188, -1.268266, -2.641385, -0.802738, 1.570796, 1.666984],accel_mss,speed_ms,0,blend_radius_m)
    movel([0.095058, -1.269118, -2.640911, -0.802360, 1.570796, 1.665855],accel_mss,speed_ms,0,blend_radius_m)
    movel([0.093443, -1.269676, -2.640600, -0.802113, 1.570796, 1.664240],accel_mss,speed_ms,0,blend_radius_m)
    movel([0.092417, -1.269568, -2.640660, -0.802161, 1.570796, 1.663213],accel_mss,speed_ms,0,blend_radius_m)
    movel([0.091928, -1.269275, -2.640823, -0.802291, 1.570796, 1.662725],accel_mss,speed_ms,0,blend_radius_m)
    movel([0.091538, -1.268021, -2.641521, -0.802847, 1.570796, 1.662334],accel_mss,speed_ms,0,blend_radius_m)
    movel([0.091986, -1.263677, -2.643923, -0.804789, 1.570796, 1.662782],accel_mss,speed_ms,0,blend_radius_m)
    movel([0.091986, -1.240641, -2.632500, -0.839248, 1.570796, 1.662782],accel_mss,speed_ms,0,blend_radius_m)
    movel([0.092892, -1.252031, -2.626355, -0.834004, 1.570796, 1.663688],accel_mss,speed_ms,0,blend_radius_m)
    movel([0.092892, -1.274936, -2.637650, -0.799803, 1.570796, 1.663688],accel_mss,speed_ms,0,blend_radius_m)
    movel([0.092456, -1.274167, -2.638083, -0.800139, 1.570796, 1.663252],accel_mss,speed_ms,0,blend_radius_m)
    movel([0.091484, -1.273582, -2.638412, -0.800395, 1.570796, 1.662280],accel_mss,speed_ms,0,blend_radius_m)
    movel([0.089925, -1.273661, -2.638368, -0.800360, 1.570796, 1.660721],accel_mss,speed_ms,0,blend_radius_m)
    movel([0.088853, -1.274032, -2.638159, -0.800198, 1.570796, 1.659650],accel_mss,speed_ms,0,blend_radius_m)
    movel([0.087200, -1.275066, -2.637577, -0.799747, 1.570796, 1.657996],accel_mss,speed_ms,0,blend_radius_m)
    movel([0.086038, -1.276387, -2.636830, -0.799172, 1.570796, 1.656834],accel_mss,speed_ms,0,blend_radius_m)
    movel([0.085412, -1.277520, -2.636188, -0.798681, 1.570796, 1.656208],accel_mss,speed_ms,0,blend_radius_m)
    movel([0.085275, -1.278937, -2.635383, -0.798069, 1.570796, 1.656071],accel_mss,speed_ms,0,blend_radius_m)
    movel([0.085716, -1.279696, -2.634950, -0.797743, 1.570796, 1.656513],accel_mss,speed_ms,0,blend_radius_m)
    movel([0.086688, -1.280271, -2.634622, -0.797496, 1.570796, 1.657485],accel_mss,speed_ms,0,blend_radius_m)
    movel([0.088237, -1.280193, -2.634667, -0.797529, 1.570796, 1.659034],accel_mss,speed_ms,0,blend_radius_m)
    movel([0.089301, -1.279828, -2.634875, -0.797686, 1.570796, 1.660098],accel_mss,speed_ms,0,blend_radius_m)
    movel([0.090946, -1.278808, -2.635456, -0.798125, 1.570796, 1.661743],accel_mss,speed_ms,0,blend_radius_m)
    movel([0.092110, -1.277495, -2.636202, -0.798692, 1.570796, 1.662906],accel_mss,speed_ms,0,blend_radius_m)
    movel([0.092743, -1.276363, -2.636843, -0.799182, 1.570796, 1.663539],accel_mss,speed_ms,0,blend_radius_m)
    movel([0.092892, -1.274936, -2.637650, -0.799803, 1.570796, 1.663688],accel_mss,speed_ms,0,blend_radius_m)
    movel([0.092892, -1.252031, -2.626355, -0.834004, 1.570796, 1.663688],accel_mss,speed_ms,0,blend_radius_m)
    movel([0.095866, -1.257950, -2.623100, -0.831339, 1.570796, 1.666662],accel_mss,speed_ms,0,blend_radius_m)
    movel([0.095866, -1.280785, -2.634329, -0.797275, 1.570796, 1.666662],accel_mss,speed_ms,0,blend_radius_m)
    movel([0.084732, -1.284577, -2.632153, -0.795659, 1.570796, 1.655528],accel_mss,speed_ms,0,blend_radius_m)
    movel([0.084732, -1.261790, -2.620966, -0.829633, 1.570796, 1.655528],accel_mss,speed_ms,0,blend_radius_m)
    movel([0.091857, -1.262078, -2.620806, -0.829506, 1.570796, 1.662654],accel_mss,speed_ms,0,blend_radius_m)
    movel([0.091857, -1.284862, -2.631989, -0.795539, 1.570796, 1.662654],accel_mss,speed_ms,0,blend_radius_m)
    movel([0.084196, -1.290169, -2.628911, -0.793309, 1.570796, 1.654992],accel_mss,speed_ms,0,blend_radius_m)
    movel([0.084196, -1.267452, -2.617787, -0.827149, 1.570796, 1.654992],accel_mss,speed_ms,0,blend_radius_m)
    movel([0.091277, -1.267753, -2.617617, -0.827018, 1.570796, 1.662073],accel_mss,speed_ms,0,blend_radius_m)
    movel([0.091277, -1.290466, -2.628737, -0.793185, 1.570796, 1.662073],accel_mss,speed_ms,0,blend_radius_m)
    movel([0.084196, -1.290169, -2.628911, -0.793309, 1.570796, 1.654992],accel_mss,speed_ms,0,blend_radius_m)
    movel([0.082180, -1.289961, -2.629032, -0.793396, 1.570796, 1.652977],accel_mss,speed_ms,0,blend_radius_m)
    movel([0.081214, -1.289396, -2.629362, -0.793632, 1.570796, 1.652010],accel_mss,speed_ms,0,blend_radius_m)
    movel([0.080773, -1.288649, -2.629796, -0.793944, 1.570796, 1.651569],accel_mss,speed_ms,0,blend_radius_m)
    movel([0.080815, -1.288184, -2.630066, -0.794139, 1.570796, 1.651612],accel_mss,speed_ms,0,blend_radius_m)
    movel([0.080815, -1.265442, -2.618920, -0.828026, 1.570796, 1.651612],accel_mss,speed_ms,0,blend_radius_m)
    movel([0.094656, -1.269337, -2.616721, -0.826331, 1.570796, 1.665452],accel_mss,speed_ms,0,blend_radius_m)
    movel([0.094656, -1.292030, -2.627823, -0.792536, 1.570796, 1.665452],accel_mss,speed_ms,0,blend_radius_m)
    movel([0.086803, -1.294654, -2.626282, -0.791453, 1.570796, 1.657599],accel_mss,speed_ms,0,blend_radius_m)
    movel([0.085190, -1.295643, -2.625698, -0.791047, 1.570796, 1.655986],accel_mss,speed_ms,0,blend_radius_m)
    movel([0.084058, -1.296915, -2.624946, -0.790527, 1.570796, 1.654854],accel_mss,speed_ms,0,blend_radius_m)
    movel([0.083405, -1.298468, -2.624026, -0.789895, 1.570796, 1.654201],accel_mss,speed_ms,0,blend_radius_m)
    movel([0.083318, -1.299383, -2.623482, -0.789524, 1.570796, 1.654114],accel_mss,speed_ms,0,blend_radius_m)
    movel([0.083707, -1.300580, -2.622769, -0.789041, 1.570796, 1.654504],accel_mss,speed_ms,0,blend_radius_m)
    movel([0.084658, -1.301145, -2.622431, -0.788813, 1.570796, 1.655454],accel_mss,speed_ms,0,blend_radius_m)
    movel([0.086171, -1.301081, -2.622469, -0.788839, 1.570796, 1.656967],accel_mss,speed_ms,0,blend_radius_m)
    movel([0.093965, -1.298501, -2.624006, -0.789882, 1.570796, 1.664761],accel_mss,speed_ms,0,blend_radius_m)
    movel([0.093965, -1.275893, -2.612976, -0.823520, 1.570796, 1.664761],accel_mss,speed_ms,0,blend_radius_m)
    movel([0.092803, -1.286986, -2.606520, -0.818883, 1.570796, 1.663599],accel_mss,speed_ms,0,blend_radius_m)
    movel([0.092803, -1.309447, -2.617426, -0.785515, 1.570796, 1.663599],accel_mss,speed_ms,0,blend_radius_m)
    movel([0.082035, -1.312966, -2.615278, -0.784145, 1.570796, 1.652832],accel_mss,speed_ms,0,blend_radius_m)
    movel([0.082035, -1.290554, -2.604411, -0.817424, 1.570796, 1.652832],accel_mss,speed_ms,0,blend_radius_m)
    movel([0.088844, -1.291815, -2.603661, -0.816912, 1.570796, 1.659641],accel_mss,speed_ms,0,blend_radius_m)
    movel([0.088844, -1.314210, -2.614514, -0.783664, 1.570796, 1.659641],accel_mss,speed_ms,0,blend_radius_m)
    movel([0.081700, -1.316541, -2.613078, -0.782769, 1.570796, 1.652496],accel_mss,speed_ms,0,blend_radius_m)
    movel([0.081700, -1.294179, -2.602251, -0.815959, 1.570796, 1.652496],accel_mss,speed_ms,0,blend_radius_m)
    movel([0.086801, -1.292488, -2.603261, -0.816640, 1.570796, 1.657598],accel_mss,speed_ms,0,blend_radius_m)
    movel([0.086801, -1.314873, -2.614107, -0.783409, 1.570796, 1.657598],accel_mss,speed_ms,0,blend_radius_m)
    movel([0.088198, -1.315719, -2.613586, -0.783084, 1.570796, 1.658994],accel_mss,speed_ms,0,blend_radius_m)
    movel([0.088617, -1.316449, -2.613136, -0.782805, 1.570796, 1.659414],accel_mss,speed_ms,0,blend_radius_m)
    movel([0.088482, -1.317788, -2.612307, -0.782294, 1.570796, 1.659278],accel_mss,speed_ms,0,blend_radius_m)
    movel([0.087883, -1.318843, -2.611653, -0.781893, 1.570796, 1.658680],accel_mss,speed_ms,0,blend_radius_m)
    movel([0.086316, -1.319779, -2.611072, -0.781538, 1.570796, 1.657112],accel_mss,speed_ms,0,blend_radius_m)
    movel([0.081244, -1.321426, -2.610046, -0.780917, 1.570796, 1.652040],accel_mss,speed_ms,0,blend_radius_m)
    movel([0.081244, -1.299133, -2.599274, -0.813983, 1.570796, 1.652040],accel_mss,speed_ms,0,blend_radius_m)
    movel([0.091252, -1.301951, -2.597565, -0.812872, 1.570796, 1.662049],accel_mss,speed_ms,0,blend_radius_m)
    movel([0.091252, -1.324205, -2.608306, -0.779878, 1.570796, 1.662049],accel_mss,speed_ms,0,blend_radius_m)
    movel([0.091345, -1.323320, -2.608862, -0.780208, 1.570796, 1.662141],accel_mss,speed_ms,0,blend_radius_m)
    movel([0.090932, -1.322594, -2.609316, -0.780479, 1.570796, 1.661728],accel_mss,speed_ms,0,blend_radius_m)
    movel([0.089460, -1.322634, -2.609291, -0.780464, 1.570796, 1.660257],accel_mss,speed_ms,0,blend_radius_m)
    movel([0.080874, -1.325395, -2.607558, -0.779436, 1.570796, 1.651670],accel_mss,speed_ms,0,blend_radius_m)
    movel([0.080874, -1.303159, -2.596830, -0.812400, 1.570796, 1.651670],accel_mss,speed_ms,0,blend_radius_m)
    movel([0.088077, -1.299501, -2.599051, -0.813837, 1.570796, 1.658874],accel_mss,speed_ms,0,blend_radius_m)
    movel([0.088077, -1.321789, -2.609819, -0.780781, 1.570796, 1.658874],accel_mss,speed_ms,0,blend_radius_m)
    movel([0.087766, -1.324885, -2.607879, -0.779625, 1.570796, 1.658562],accel_mss,speed_ms,0,blend_radius_m)
    movel([0.087766, -1.302641, -2.597146, -0.812602, 1.570796, 1.658562],accel_mss,speed_ms,0,blend_radius_m)
    movel([0.087280, -1.307547, -2.594144, -0.810698, 1.570796, 1.658076],accel_mss,speed_ms,0,blend_radius_m)
    movel([0.087280, -1.329720, -2.604824, -0.777845, 1.570796, 1.658076],accel_mss,speed_ms,0,blend_radius_m)
    movel([0.086866, -1.329003, -2.605279, -0.778107, 1.570796, 1.657662],accel_mss,speed_ms,0,blend_radius_m)
    movel([0.085949, -1.328445, -2.605632, -0.778312, 1.570796, 1.656745],accel_mss,speed_ms,0,blend_radius_m)
    movel([0.084484, -1.328488, -2.605605, -0.778296, 1.570796, 1.655281],accel_mss,speed_ms,0,blend_radius_m)
    movel([0.083479, -1.328809, -2.605401, -0.778178, 1.570796, 1.654276],accel_mss,speed_ms,0,blend_radius_m)
    movel([0.081932, -1.329730, -2.604817, -0.777842, 1.570796, 1.652728],accel_mss,speed_ms,0,blend_radius_m)
    movel([0.080847, -1.330926, -2.604057, -0.777407, 1.570796, 1.651643],accel_mss,speed_ms,0,blend_radius_m)
    movel([0.080265, -1.331958, -2.603398, -0.777032, 1.570796, 1.651062],accel_mss,speed_ms,0,blend_radius_m)
    movel([0.080145, -1.333263, -2.602565, -0.776561, 1.570796, 1.650941],accel_mss,speed_ms,0,blend_radius_m)
    movel([0.080564, -1.333972, -2.602111, -0.776307, 1.570796, 1.651360],accel_mss,speed_ms,0,blend_radius_m)
    movel([0.081481, -1.334521, -2.601759, -0.776110, 1.570796, 1.652277],accel_mss,speed_ms,0,blend_radius_m)
    movel([0.082937, -1.334478, -2.601786, -0.776125, 1.570796, 1.653733],accel_mss,speed_ms,0,blend_radius_m)
    movel([0.083935, -1.334161, -2.601989, -0.776239, 1.570796, 1.654731],accel_mss,speed_ms,0,blend_radius_m)
    movel([0.085475, -1.333252, -2.602572, -0.776565, 1.570796, 1.656271],accel_mss,speed_ms,0,blend_radius_m)
    movel([0.086561, -1.332064, -2.603331, -0.776994, 1.570796, 1.657357],accel_mss,speed_ms,0,blend_radius_m)
    movel([0.087149, -1.331032, -2.603989, -0.777368, 1.570796, 1.657945],accel_mss,speed_ms,0,blend_radius_m)
    movel([0.087280, -1.329720, -2.604824, -0.777845, 1.570796, 1.658076],accel_mss,speed_ms,0,blend_radius_m)
    movel([0.087280, -1.307547, -2.594144, -0.810698, 1.570796, 1.658076],accel_mss,speed_ms,0,blend_radius_m)
    movel([0.089398, -1.320100, -2.586322, -0.805968, 1.570796, 1.660194],accel_mss,speed_ms,0,blend_radius_m)
    movel([0.089398, -1.342088, -2.596863, -0.773437, 1.570796, 1.660194],accel_mss,speed_ms,0,blend_radius_m)
    movel([0.079037, -1.345319, -2.594750, -0.772320, 1.570796, 1.649833],accel_mss,speed_ms,0,blend_radius_m)
    movel([0.079037, -1.323379, -2.584244, -0.804766, 1.570796, 1.649833],accel_mss,speed_ms,0,blend_radius_m)
    movel([0.089398, -1.320100, -2.586322, -0.805968, 1.570796, 1.660194],accel_mss,speed_ms,0,blend_radius_m)
    movel([0.089398, -1.342088, -2.596863, -0.773437, 1.570796, 1.660194],accel_mss,speed_ms,0,blend_radius_m)
    movel([0.089089, -1.345094, -2.594898, -0.772398, 1.570796, 1.659885],accel_mss,speed_ms,0,blend_radius_m)
    movel([0.088466, -1.346528, -2.593955, -0.771906, 1.570796, 1.659262],accel_mss,speed_ms,0,blend_radius_m)
    movel([0.087397, -1.347683, -2.593194, -0.771512, 1.570796, 1.658193],accel_mss,speed_ms,0,blend_radius_m)
    movel([0.086372, -1.348411, -2.592713, -0.771265, 1.570796, 1.657169],accel_mss,speed_ms,0,blend_radius_m)
    movel([0.084859, -1.349289, -2.592132, -0.770967, 1.570796, 1.655656],accel_mss,speed_ms,0,blend_radius_m)
    movel([0.082410, -1.350047, -2.591631, -0.770712, 1.570796, 1.653206],accel_mss,speed_ms,0,blend_radius_m)
    movel([0.080981, -1.350079, -2.591610, -0.770701, 1.570796, 1.651777],accel_mss,speed_ms,0,blend_radius_m)
    movel([0.080040, -1.349960, -2.591688, -0.770741, 1.570796, 1.650837],accel_mss,speed_ms,0,blend_radius_m)
    movel([0.079139, -1.349418, -2.592047, -0.770924, 1.570796, 1.649935],accel_mss,speed_ms,0,blend_radius_m)
    movel([0.078764, -1.348299, -2.592787, -0.771303, 1.570796, 1.649561],accel_mss,speed_ms,0,blend_radius_m)
    movel([0.079037, -1.345319, -2.594750, -0.772320, 1.570796, 1.649833],accel_mss,speed_ms,0,blend_radius_m)
    movel([0.079037, -1.323379, -2.584244, -0.804766, 1.570796, 1.649833],accel_mss,speed_ms,0,blend_radius_m)
    movel([0.084601, -1.334987, -2.576777, -0.800625, 1.570796, 1.655398],accel_mss,speed_ms,0,blend_radius_m)
    movel([0.084601, -1.356749, -2.587156, -0.768484, 1.570796, 1.655398],accel_mss,speed_ms,0,blend_radius_m)
    movel([0.077808, -1.358834, -2.585751, -0.767804, 1.570796, 1.648604],accel_mss,speed_ms,0,blend_radius_m)
    movel([0.077808, -1.337105, -2.575395, -0.799889, 1.570796, 1.648604],accel_mss,speed_ms,0,blend_radius_m)
    movel([0.083145, -1.335439, -2.576483, -0.800468, 1.570796, 1.653941],accel_mss,speed_ms,0,blend_radius_m)
    movel([0.083145, -1.357194, -2.586857, -0.768338, 1.570796, 1.653941],accel_mss,speed_ms,0,blend_radius_m)
    movel([0.084198, -1.356056, -2.587621, -0.768711, 1.570796, 1.654994],accel_mss,speed_ms,0,blend_radius_m)
    movel([0.084766, -1.355065, -2.588286, -0.769038, 1.570796, 1.655563],accel_mss,speed_ms,0,blend_radius_m)
    movel([0.084891, -1.353800, -2.589133, -0.769457, 1.570796, 1.655687],accel_mss,speed_ms,0,blend_radius_m)
    movel([0.084486, -1.353104, -2.589597, -0.769688, 1.570796, 1.655282],accel_mss,speed_ms,0,blend_radius_m)
    movel([0.083592, -1.352558, -2.589961, -0.769869, 1.570796, 1.654388],accel_mss,speed_ms,0,blend_radius_m)
    movel([0.082168, -1.352587, -2.589942, -0.769860, 1.570796, 1.652964],accel_mss,speed_ms,0,blend_radius_m)
    movel([0.081191, -1.352889, -2.589741, -0.769759, 1.570796, 1.651988],accel_mss,speed_ms,0,blend_radius_m)
    movel([0.079688, -1.353765, -2.589156, -0.769468, 1.570796, 1.650485],accel_mss,speed_ms,0,blend_radius_m)
    movel([0.078636, -1.354909, -2.588390, -0.769089, 1.570796, 1.649433],accel_mss,speed_ms,0,blend_radius_m)
    movel([0.078073, -1.355901, -2.587726, -0.768762, 1.570796, 1.648869],accel_mss,speed_ms,0,blend_radius_m)
    movel([0.077959, -1.357160, -2.586880, -0.768350, 1.570796, 1.648755],accel_mss,speed_ms,0,blend_radius_m)
    movel([0.078369, -1.357847, -2.586417, -0.768125, 1.570796, 1.649165],accel_mss,speed_ms,0,blend_radius_m)
    movel([0.079262, -1.358385, -2.586054, -0.767950, 1.570796, 1.650059],accel_mss,speed_ms,0,blend_radius_m)
    movel([0.079262, -1.336649, -2.575693, -0.800047, 1.570796, 1.650059],accel_mss,speed_ms,0,blend_radius_m)
    movel([0.084355, -1.337545, -2.575108, -0.799737, 1.570796, 1.655151],accel_mss,speed_ms,0,blend_radius_m)
    movel([0.084355, -1.359267, -2.585459, -0.767663, 1.570796, 1.655151],accel_mss,speed_ms,0,blend_radius_m)
    movel([0.077357, -1.363833, -2.582358, -0.766198, 1.570796, 1.648153],accel_mss,speed_ms,0,blend_radius_m)
    movel([0.077357, -1.342184, -2.572057, -0.798148, 1.570796, 1.648153],accel_mss,speed_ms,0,blend_radius_m)
    movel([0.083866, -1.342631, -2.571761, -0.797996, 1.570796, 1.654663],accel_mss,speed_ms,0,blend_radius_m)
    movel([0.083866, -1.364274, -2.582058, -0.766058, 1.570796, 1.654663],accel_mss,speed_ms,0,blend_radius_m)
    movel([0.077357, -1.363833, -2.582358, -0.766198, 1.570796, 1.648153],accel_mss,speed_ms,0,blend_radius_m)
    movel([0.075502, -1.363596, -2.582520, -0.766273, 1.570796, 1.646299],accel_mss,speed_ms,0,blend_radius_m)
    movel([0.074611, -1.363065, -2.582882, -0.766442, 1.570796, 1.645407],accel_mss,speed_ms,0,blend_radius_m)
    movel([0.074200, -1.362384, -2.583345, -0.766660, 1.570796, 1.644996],accel_mss,speed_ms,0,blend_radius_m)
    movel([0.074236, -1.361969, -2.583628, -0.766793, 1.570796, 1.645032],accel_mss,speed_ms,0,blend_radius_m)
    movel([0.074236, -1.340289, -2.573306, -0.798793, 1.570796, 1.645032],accel_mss,speed_ms,0,blend_radius_m)
    movel([0.083938, -1.351574, -2.565794, -0.795021, 1.570796, 1.654734],accel_mss,speed_ms,0,blend_radius_m)
    movel([0.083938, -1.373074, -2.575994, -0.763322, 1.570796, 1.654734],accel_mss,speed_ms,0,blend_radius_m)
    movel([0.084415, -1.372932, -2.576092, -0.763365, 1.570796, 1.655211],accel_mss,speed_ms,0,blend_radius_m)
    movel([0.085327, -1.373060, -2.576003, -0.763326, 1.570796, 1.656123],accel_mss,speed_ms,0,blend_radius_m)
    movel([0.085762, -1.373330, -2.575815, -0.763244, 1.570796, 1.656558],accel_mss,speed_ms,0,blend_radius_m)
    movel([0.086156, -1.374011, -2.575341, -0.763037, 1.570796, 1.656952],accel_mss,speed_ms,0,blend_radius_m)
    movel([0.085992, -1.375649, -2.574198, -0.762542, 1.570796, 1.656788],accel_mss,speed_ms,0,blend_radius_m)
    movel([0.085436, -1.376606, -2.573528, -0.762254, 1.570796, 1.656232],accel_mss,speed_ms,0,blend_radius_m)
    movel([0.084921, -1.377154, -2.573145, -0.762091, 1.570796, 1.655718],accel_mss,speed_ms,0,blend_radius_m)
    movel([0.083934, -1.377840, -2.572663, -0.761886, 1.570796, 1.654730],accel_mss,speed_ms,0,blend_radius_m)
    movel([0.082987, -1.378120, -2.572467, -0.761803, 1.570796, 1.653783],accel_mss,speed_ms,0,blend_radius_m)
    movel([0.082079, -1.377992, -2.572556, -0.761841, 1.570796, 1.652875],accel_mss,speed_ms,0,blend_radius_m)
    movel([0.080735, -1.377599, -2.572832, -0.761958, 1.570796, 1.651531],accel_mss,speed_ms,0,blend_radius_m)
    movel([0.076361, -1.374945, -2.574690, -0.762754, 1.570796, 1.647158],accel_mss,speed_ms,0,blend_radius_m)
    movel([0.075855, -1.380636, -2.570695, -0.761059, 1.570796, 1.646652],accel_mss,speed_ms,0,blend_radius_m)
    movel([0.075855, -1.359260, -2.560578, -0.792551, 1.570796, 1.646652],accel_mss,speed_ms,0,blend_radius_m)
    movel([0.085302, -1.361226, -2.559231, -0.791932, 1.570796, 1.656098],accel_mss,speed_ms,0,blend_radius_m)
    movel([0.085302, -1.382569, -2.569327, -0.760493, 1.570796, 1.656098],accel_mss,speed_ms,0,blend_radius_m)
    movel([0.084951, -1.381490, -2.570090, -0.760808, 1.570796, 1.655748],accel_mss,speed_ms,0,blend_radius_m)
    movel([0.083616, -1.381093, -2.570371, -0.760925, 1.570796, 1.654412],accel_mss,speed_ms,0,blend_radius_m)
    movel([0.081297, -1.381381, -2.570168, -0.760840, 1.570796, 1.652093],accel_mss,speed_ms,0,blend_radius_m)
    movel([0.079882, -1.381799, -2.569872, -0.760718, 1.570796, 1.650678],accel_mss,speed_ms,0,blend_radius_m)
    movel([0.077488, -1.382902, -2.569091, -0.760397, 1.570796, 1.648285],accel_mss,speed_ms,0,blend_radius_m)
    movel([0.076004, -1.384128, -2.568219, -0.760041, 1.570796, 1.646800],accel_mss,speed_ms,0,blend_radius_m)
    movel([0.075427, -1.385475, -2.567260, -0.759654, 1.570796, 1.646223],accel_mss,speed_ms,0,blend_radius_m)
    movel([0.075356, -1.386279, -2.566687, -0.759423, 1.570796, 1.646153],accel_mss,speed_ms,0,blend_radius_m)
    movel([0.075719, -1.387343, -2.565926, -0.759120, 1.570796, 1.646515],accel_mss,speed_ms,0,blend_radius_m)
    movel([0.077052, -1.387729, -2.565650, -0.759011, 1.570796, 1.647848],accel_mss,speed_ms,0,blend_radius_m)
    movel([0.079357, -1.387440, -2.565856, -0.759093, 1.570796, 1.650153],accel_mss,speed_ms,0,blend_radius_m)
    movel([0.080762, -1.387029, -2.566151, -0.759210, 1.570796, 1.651558],accel_mss,speed_ms,0,blend_radius_m)
    movel([0.083144, -1.385942, -2.566927, -0.759520, 1.570796, 1.653941],accel_mss,speed_ms,0,blend_radius_m)
    movel([0.084631, -1.384727, -2.567794, -0.759869, 1.570796, 1.655428],accel_mss,speed_ms,0,blend_radius_m)
    movel([0.085221, -1.383378, -2.568752, -0.760258, 1.570796, 1.656018],accel_mss,speed_ms,0,blend_radius_m)
    movel([0.085302, -1.382569, -2.569327, -0.760493, 1.570796, 1.656098],accel_mss,speed_ms,0,blend_radius_m)
    movel([0.085302, -1.361226, -2.559231, -0.791932, 1.570796, 1.656098],accel_mss,speed_ms,0,blend_radius_m)
    movel([0.082366, -1.368061, -2.554506, -0.789822, 1.570796, 1.653162],accel_mss,speed_ms,0,blend_radius_m)
    movel([0.082366, -1.389292, -2.564528, -0.758569, 1.570796, 1.653162],accel_mss,speed_ms,0,blend_radius_m)
    movel([0.082833, -1.389156, -2.564625, -0.758607, 1.570796, 1.653629],accel_mss,speed_ms,0,blend_radius_m)
    movel([0.083728, -1.389287, -2.564532, -0.758571, 1.570796, 1.654525],accel_mss,speed_ms,0,blend_radius_m)
    movel([0.084156, -1.389553, -2.564341, -0.758496, 1.570796, 1.654952],accel_mss,speed_ms,0,blend_radius_m)
    movel([0.084544, -1.390219, -2.563861, -0.758309, 1.570796, 1.655340],accel_mss,speed_ms,0,blend_radius_m)
    movel([0.084386, -1.391819, -2.562707, -0.757863, 1.570796, 1.655182],accel_mss,speed_ms,0,blend_radius_m)
    movel([0.083842, -1.392751, -2.562034, -0.757605, 1.570796, 1.654638],accel_mss,speed_ms,0,blend_radius_m)
    movel([0.083338, -1.393283, -2.561648, -0.757458, 1.570796, 1.654134],accel_mss,speed_ms,0,blend_radius_m)
    movel([0.082370, -1.393949, -2.561166, -0.757275, 1.570796, 1.653166],accel_mss,speed_ms,0,blend_radius_m)
    movel([0.081441, -1.394216, -2.560972, -0.757201, 1.570796, 1.652237],accel_mss,speed_ms,0,blend_radius_m)
    movel([0.080550, -1.394087, -2.561065, -0.757237, 1.570796, 1.651346],accel_mss,speed_ms,0,blend_radius_m)
    movel([0.079230, -1.393696, -2.561349, -0.757344, 1.570796, 1.650026],accel_mss,speed_ms,0,blend_radius_m)
    movel([0.074934, -1.391078, -2.563242, -0.758069, 1.570796, 1.645730],accel_mss,speed_ms,0,blend_radius_m)
    movel([0.074447, -1.396636, -2.559211, -0.756542, 1.570796, 1.645243],accel_mss,speed_ms,0,blend_radius_m)
    movel([0.074447, -1.375530, -2.549268, -0.787590, 1.570796, 1.645243],accel_mss,speed_ms,0,blend_radius_m)
    movel([0.083877, -1.375892, -2.549012, -0.787484, 1.570796, 1.654673],accel_mss,speed_ms,0,blend_radius_m)
    movel([0.083877, -1.396992, -2.558951, -0.756446, 1.570796, 1.654673],accel_mss,speed_ms,0,blend_radius_m)
    movel([0.083451, -1.401339, -2.555765, -0.755285, 1.570796, 1.654248],accel_mss,speed_ms,0,blend_radius_m)
    movel([0.079991, -1.400025, -2.556731, -0.755633, 1.570796, 1.650788],accel_mss,speed_ms,0,blend_radius_m)
    movel([0.079880, -1.401207, -2.555862, -0.755320, 1.570796, 1.650677],accel_mss,speed_ms,0,blend_radius_m)
    movel([0.079347, -1.402125, -2.555186, -0.755078, 1.570796, 1.650143],accel_mss,speed_ms,0,blend_radius_m)
    movel([0.078850, -1.402650, -2.554799, -0.754941, 1.570796, 1.649647],accel_mss,speed_ms,0,blend_radius_m)
    movel([0.077436, -1.403438, -2.554217, -0.754735, 1.570796, 1.648232],accel_mss,speed_ms,0,blend_radius_m)
    movel([0.076517, -1.403702, -2.554021, -0.754666, 1.570796, 1.647313],accel_mss,speed_ms,0,blend_radius_m)
    movel([0.075174, -1.403708, -2.554017, -0.754664, 1.570796, 1.645970],accel_mss,speed_ms,0,blend_radius_m)
    movel([0.074324, -1.403191, -2.554399, -0.754799, 1.570796, 1.645120],accel_mss,speed_ms,0,blend_radius_m)
    movel([0.073966, -1.402149, -2.555168, -0.755072, 1.570796, 1.644762],accel_mss,speed_ms,0,blend_radius_m)
    movel([0.074068, -1.400971, -2.556036, -0.755382, 1.570796, 1.644865],accel_mss,speed_ms,0,blend_radius_m)
    movel([0.074633, -1.399657, -2.557001, -0.755731, 1.570796, 1.645429],accel_mss,speed_ms,0,blend_radius_m)
    movel([0.075129, -1.399128, -2.557389, -0.755872, 1.570796, 1.645925],accel_mss,speed_ms,0,blend_radius_m)
    movel([0.076088, -1.398465, -2.557875, -0.756049, 1.570796, 1.646885],accel_mss,speed_ms,0,blend_radius_m)
    movel([0.076088, -1.377391, -2.547951, -0.787047, 1.570796, 1.646885],accel_mss,speed_ms,0,blend_radius_m)
    movel([0.067435, -1.341079, -2.572786, -0.798524, 1.570796, 1.638231],accel_mss,speed_ms,0,blend_radius_m)
    movel([0.067435, -1.362745, -2.583099, -0.766544, 1.570796, 1.638231],accel_mss,speed_ms,0,blend_radius_m)
    movel([0.061103, -1.364759, -2.581726, -0.765904, 1.570796, 1.631900],accel_mss,speed_ms,0,blend_radius_m)
    movel([0.061103, -1.343125, -2.571435, -0.797829, 1.570796, 1.631900],accel_mss,speed_ms,0,blend_radius_m)
    movel([0.064418, -1.342050, -2.572145, -0.798194, 1.570796, 1.635214],accel_mss,speed_ms,0,blend_radius_m)
    movel([0.064418, -1.363701, -2.582448, -0.766240, 1.570796, 1.635214],accel_mss,speed_ms,0,blend_radius_m)
    movel([0.064982, -1.364026, -2.582226, -0.766136, 1.570796, 1.635778],accel_mss,speed_ms,0,blend_radius_m)
    movel([0.065244, -1.364447, -2.581939, -0.766003, 1.570796, 1.636040],accel_mss,speed_ms,0,blend_radius_m)
    movel([0.065185, -1.365220, -2.581410, -0.765758, 1.570796, 1.635981],accel_mss,speed_ms,0,blend_radius_m)
    movel([0.064845, -1.365831, -2.580992, -0.765566, 1.570796, 1.635641],accel_mss,speed_ms,0,blend_radius_m)
    movel([0.064205, -1.366536, -2.580509, -0.765344, 1.570796, 1.635001],accel_mss,speed_ms,0,blend_radius_m)
    movel([0.063285, -1.367078, -2.580137, -0.765174, 1.570796, 1.634081],accel_mss,speed_ms,0,blend_radius_m)
    movel([0.062684, -1.367269, -2.580006, -0.765114, 1.570796, 1.633480],accel_mss,speed_ms,0,blend_radius_m)
    movel([0.061802, -1.367299, -2.579985, -0.765105, 1.570796, 1.632598],accel_mss,speed_ms,0,blend_radius_m)
    movel([0.061238, -1.366977, -2.580207, -0.765206, 1.570796, 1.632035],accel_mss,speed_ms,0,blend_radius_m)
    movel([0.060975, -1.366559, -2.580493, -0.765337, 1.570796, 1.631771],accel_mss,speed_ms,0,blend_radius_m)
    movel([0.061030, -1.365788, -2.581022, -0.765579, 1.570796, 1.631826],accel_mss,speed_ms,0,blend_radius_m)
    movel([0.061368, -1.365177, -2.581440, -0.765772, 1.570796, 1.632164],accel_mss,speed_ms,0,blend_radius_m)
    movel([0.062007, -1.364470, -2.581923, -0.765996, 1.570796, 1.632803],accel_mss,speed_ms,0,blend_radius_m)
    movel([0.062007, -1.342831, -2.571629, -0.797929, 1.570796, 1.632803],accel_mss,speed_ms,0,blend_radius_m)
    movel([0.064989, -1.346207, -2.569388, -0.796794, 1.570796, 1.635786],accel_mss,speed_ms,0,blend_radius_m)
    movel([0.064989, -1.367793, -2.579646, -0.764951, 1.570796, 1.635786],accel_mss,speed_ms,0,blend_radius_m)
    movel([0.060682, -1.370655, -2.577671, -0.764063, 1.570796, 1.631479],accel_mss,speed_ms,0,blend_radius_m)
    movel([0.060682, -1.349116, -2.567445, -0.795828, 1.570796, 1.631479],accel_mss,speed_ms,0,blend_radius_m)
    movel([0.064756, -1.349331, -2.567301, -0.795757, 1.570796, 1.635552],accel_mss,speed_ms,0,blend_radius_m)
    movel([0.064756, -1.370866, -2.577525, -0.763998, 1.570796, 1.635552],accel_mss,speed_ms,0,blend_radius_m)
    movel([0.060682, -1.370655, -2.577671, -0.764063, 1.570796, 1.631479],accel_mss,speed_ms,0,blend_radius_m)
    movel([0.059522, -1.370525, -2.577761, -0.764103, 1.570796, 1.630318],accel_mss,speed_ms,0,blend_radius_m)
    movel([0.058959, -1.370206, -2.577982, -0.764201, 1.570796, 1.629755],accel_mss,speed_ms,0,blend_radius_m)
    movel([0.058695, -1.369791, -2.578268, -0.764330, 1.570796, 1.629491],accel_mss,speed_ms,0,blend_radius_m)
    movel([0.058713, -1.369535, -2.578445, -0.764409, 1.570796, 1.629509],accel_mss,speed_ms,0,blend_radius_m)
    movel([0.058713, -1.347978, -2.568206, -0.796205, 1.570796, 1.629509],accel_mss,speed_ms,0,blend_radius_m)
    movel([0.066313, -1.355654, -2.563035, -0.793700, 1.570796, 1.637109],accel_mss,speed_ms,0,blend_radius_m)
    movel([0.066313, -1.377088, -2.573191, -0.762110, 1.570796, 1.637109],accel_mss,speed_ms,0,blend_radius_m)
    movel([0.060232, -1.377007, -2.573247, -0.762135, 1.570796, 1.631028],accel_mss,speed_ms,0,blend_radius_m)
    movel([0.060232, -1.355572, -2.563091, -0.793726, 1.570796, 1.631028],accel_mss,speed_ms,0,blend_radius_m)
    movel([0.066313, -1.355654, -2.563035, -0.793700, 1.570796, 1.637109],accel_mss,speed_ms,0,blend_radius_m)
    movel([0.066313, -1.377088, -2.573191, -0.762110, 1.570796, 1.637109],accel_mss,speed_ms,0,blend_radius_m)
    movel([0.059947, -1.381041, -2.570408, -0.760940, 1.570796, 1.630743],accel_mss,speed_ms,0,blend_radius_m)
    movel([0.059947, -1.359673, -2.560296, -0.792421, 1.570796, 1.630743],accel_mss,speed_ms,0,blend_radius_m)
    movel([0.062254, -1.355681, -2.563017, -0.793691, 1.570796, 1.633051],accel_mss,speed_ms,0,blend_radius_m)
    movel([0.062254, -1.377114, -2.573172, -0.762103, 1.570796, 1.633051],accel_mss,speed_ms,0,blend_radius_m)
    movel([0.062070, -1.379640, -2.571397, -0.761352, 1.570796, 1.632866],accel_mss,speed_ms,0,blend_radius_m)
    movel([0.062070, -1.358248, -2.561269, -0.792872, 1.570796, 1.632866],accel_mss,speed_ms,0,blend_radius_m)
    movel([0.066057, -1.358995, -2.560759, -0.792635, 1.570796, 1.636854],accel_mss,speed_ms,0,blend_radius_m)
    movel([0.066057, -1.380374, -2.570879, -0.761136, 1.570796, 1.636854],accel_mss,speed_ms,0,blend_radius_m)
    movel([0.059858, -1.382297, -2.569519, -0.760573, 1.570796, 1.630654],accel_mss,speed_ms,0,blend_radius_m)
    movel([0.059858, -1.360950, -2.559421, -0.792019, 1.570796, 1.630654],accel_mss,speed_ms,0,blend_radius_m)
    movel([0.065901, -1.361042, -2.559357, -0.791990, 1.570796, 1.636698],accel_mss,speed_ms,0,blend_radius_m)
    movel([0.065901, -1.382388, -2.569455, -0.760546, 1.570796, 1.636698],accel_mss,speed_ms,0,blend_radius_m)
    movel([0.059717, -1.384301, -2.568096, -0.759991, 1.570796, 1.630513],accel_mss,speed_ms,0,blend_radius_m)
    movel([0.059717, -1.362987, -2.558019, -0.791382, 1.570796, 1.630513],accel_mss,speed_ms,0,blend_radius_m)
    movel([0.065901, -1.361042, -2.559357, -0.791990, 1.570796, 1.636698],accel_mss,speed_ms,0,blend_radius_m)
    movel([0.065901, -1.382388, -2.569455, -0.760546, 1.570796, 1.636698],accel_mss,speed_ms,0,blend_radius_m)
    movel([0.065727, -1.384648, -2.567850, -0.759891, 1.570796, 1.636523],accel_mss,speed_ms,0,blend_radius_m)
    movel([0.065375, -1.385489, -2.567250, -0.759650, 1.570796, 1.636171],accel_mss,speed_ms,0,blend_radius_m)
    movel([0.065062, -1.385829, -2.567008, -0.759552, 1.570796, 1.635859],accel_mss,speed_ms,0,blend_radius_m)
    movel([0.064456, -1.386259, -2.566701, -0.759429, 1.570796, 1.635253],accel_mss,speed_ms,0,blend_radius_m)
    movel([0.063870, -1.386439, -2.566572, -0.759378, 1.570796, 1.634666],accel_mss,speed_ms,0,blend_radius_m)
    movel([0.063301, -1.386370, -2.566622, -0.759398, 1.570796, 1.634098],accel_mss,speed_ms,0,blend_radius_m)
    movel([0.063026, -1.386210, -2.566736, -0.759443, 1.570796, 1.633823],accel_mss,speed_ms,0,blend_radius_m)
    movel([0.062788, -1.385551, -2.567207, -0.759632, 1.570796, 1.633585],accel_mss,speed_ms,0,blend_radius_m)
    movel([0.062955, -1.383297, -2.568810, -0.760282, 1.570796, 1.633751],accel_mss,speed_ms,0,blend_radius_m)
    movel([0.062955, -1.361966, -2.558723, -0.791701, 1.570796, 1.633751],accel_mss,speed_ms,0,blend_radius_m)
    movel([0.062825, -1.363749, -2.557494, -0.791146, 1.570796, 1.633622],accel_mss,speed_ms,0,blend_radius_m)
    movel([0.062825, -1.385050, -2.567563, -0.759776, 1.570796, 1.633622],accel_mss,speed_ms,0,blend_radius_m)
    movel([0.059472, -1.387795, -2.565602, -0.758992, 1.570796, 1.630268],accel_mss,speed_ms,0,blend_radius_m)
    movel([0.059472, -1.366540, -2.555563, -0.790286, 1.570796, 1.630268],accel_mss,speed_ms,0,blend_radius_m)
    movel([0.065190, -1.370438, -2.552847, -0.789103, 1.570796, 1.635986],accel_mss,speed_ms,0,blend_radius_m)
    movel([0.065190, -1.391629, -2.562844, -0.757915, 1.570796, 1.635986],accel_mss,speed_ms,0,blend_radius_m)
    movel([0.059073, -1.393497, -2.561493, -0.757399, 1.570796, 1.629870],accel_mss,speed_ms,0,blend_radius_m)
    movel([0.058867, -1.396453, -2.559345, -0.756592, 1.570796, 1.629664],accel_mss,speed_ms,0,blend_radius_m)
    movel([0.058867, -1.375344, -2.549400, -0.787645, 1.570796, 1.629664],accel_mss,speed_ms,0,blend_radius_m)
    movel([0.064774, -1.375967, -2.548960, -0.787462, 1.570796, 1.635570],accel_mss,speed_ms,0,blend_radius_m)
    movel([0.064774, -1.397065, -2.558898, -0.756426, 1.570796, 1.635570],accel_mss,speed_ms,0,blend_radius_m)
    movel([0.058833, -1.396944, -2.558986, -0.756459, 1.570796, 1.629630],accel_mss,speed_ms,0,blend_radius_m)
    movel([0.058833, -1.375844, -2.549047, -0.787498, 1.570796, 1.629630],accel_mss,speed_ms,0,blend_radius_m)
    movel([0.064774, -1.375967, -2.548960, -0.787462, 1.570796, 1.635570],accel_mss,speed_ms,0,blend_radius_m)
    movel([0.064774, -1.397065, -2.558898, -0.756426, 1.570796, 1.635570],accel_mss,speed_ms,0,blend_radius_m)
    movel([0.058561, -1.400863, -2.556115, -0.755411, 1.570796, 1.629358],accel_mss,speed_ms,0,blend_radius_m)
    movel([0.058561, -1.379830, -2.546218, -0.786341, 1.570796, 1.629358],accel_mss,speed_ms,0,blend_radius_m)
    movel([0.060809, -1.375964, -2.548961, -0.787463, 1.570796, 1.631606],accel_mss,speed_ms,0,blend_radius_m)
    movel([0.060809, -1.397062, -2.558900, -0.756427, 1.570796, 1.631606],accel_mss,speed_ms,0,blend_radius_m)
    movel([0.060633, -1.399516, -2.557105, -0.755768, 1.570796, 1.631430],accel_mss,speed_ms,0,blend_radius_m)
    movel([0.060633, -1.378460, -2.547193, -0.786736, 1.570796, 1.631430],accel_mss,speed_ms,0,blend_radius_m)
    movel([0.064530, -1.379214, -2.546657, -0.786519, 1.570796, 1.635327],accel_mss,speed_ms,0,blend_radius_m)
    movel([0.064530, -1.400257, -2.556561, -0.755571, 1.570796, 1.635327],accel_mss,speed_ms,0,blend_radius_m)
    movel([0.058477, -1.402083, -2.555217, -0.755089, 1.570796, 1.629273],accel_mss,speed_ms,0,blend_radius_m)
    movel([0.058477, -1.381071, -2.545332, -0.785985, 1.570796, 1.629273],accel_mss,speed_ms,0,blend_radius_m)
    movel([0.064530, -1.379214, -2.546657, -0.786519, 1.570796, 1.635327],accel_mss,speed_ms,0,blend_radius_m)
    movel([0.064530, -1.400257, -2.556561, -0.755571, 1.570796, 1.635327],accel_mss,speed_ms,0,blend_radius_m)
    movel([0.064363, -1.402459, -2.554940, -0.754991, 1.570796, 1.635159],accel_mss,speed_ms,0,blend_radius_m)
    movel([0.064020, -1.403276, -2.554336, -0.754777, 1.570796, 1.634816],accel_mss,speed_ms,0,blend_radius_m)
    movel([0.063714, -1.403606, -2.554092, -0.754691, 1.570796, 1.634510],accel_mss,speed_ms,0,blend_radius_m)
    movel([0.063121, -1.404021, -2.553785, -0.754583, 1.570796, 1.633918],accel_mss,speed_ms,0,blend_radius_m)
    movel([0.062547, -1.404193, -2.553658, -0.754538, 1.570796, 1.633343],accel_mss,speed_ms,0,blend_radius_m)
    movel([0.061990, -1.404122, -2.553710, -0.754557, 1.570796, 1.632787],accel_mss,speed_ms,0,blend_radius_m)
    movel([0.061721, -1.403965, -2.553827, -0.754598, 1.570796, 1.632517],accel_mss,speed_ms,0,blend_radius_m)
    movel([0.061487, -1.403320, -2.554303, -0.754765, 1.570796, 1.632283],accel_mss,speed_ms,0,blend_radius_m)
    movel([0.061487, -1.382330, -2.544432, -0.785627, 1.570796, 1.632283],accel_mss,speed_ms,0,blend_radius_m)
    movel([0.061646, -1.380096, -2.546029, -0.786265, 1.570796, 1.632443],accel_mss,speed_ms,0,blend_radius_m)
    movel([0.061646, -1.401124, -2.555923, -0.755342, 1.570796, 1.632443],accel_mss,speed_ms,0,blend_radius_m)
    movel([0.061487, -1.403320, -2.554303, -0.754765, 1.570796, 1.632283],accel_mss,speed_ms,0,blend_radius_m)
    movel([0.061146, -1.404137, -2.553699, -0.754553, 1.570796, 1.631943],accel_mss,speed_ms,0,blend_radius_m)
    movel([0.060842, -1.404467, -2.553455, -0.754467, 1.570796, 1.631638],accel_mss,speed_ms,0,blend_radius_m)
    movel([0.060250, -1.404883, -2.553147, -0.754360, 1.570796, 1.631047],accel_mss,speed_ms,0,blend_radius_m)
    movel([0.059389, -1.405142, -2.552955, -0.754293, 1.570796, 1.630186],accel_mss,speed_ms,0,blend_radius_m)
    movel([0.058832, -1.405072, -2.553006, -0.754311, 1.570796, 1.629629],accel_mss,speed_ms,0,blend_radius_m)
    movel([0.058563, -1.404916, -2.553122, -0.754351, 1.570796, 1.629359],accel_mss,speed_ms,0,blend_radius_m)
    movel([0.058326, -1.404274, -2.553598, -0.754517, 1.570796, 1.629122],accel_mss,speed_ms,0,blend_radius_m)
    movel([0.058477, -1.402083, -2.555217, -0.755089, 1.570796, 1.629273],accel_mss,speed_ms,0,blend_radius_m)
    movel([0.058477, -1.381071, -2.545332, -0.785985, 1.570796, 1.629273],accel_mss,speed_ms,0,blend_radius_m)
    movel([0.063848, -1.388375, -2.540078, -0.783935, 1.570796, 1.634644],accel_mss,speed_ms,0,blend_radius_m)
    movel([0.063848, -1.409262, -2.549885, -0.753241, 1.570796, 1.634644],accel_mss,speed_ms,0,blend_radius_m)
    movel([0.057860, -1.411046, -2.548549, -0.752794, 1.570796, 1.628656],accel_mss,speed_ms,0,blend_radius_m)
    movel([0.057860, -1.390190, -2.538761, -0.783438, 1.570796, 1.628656],accel_mss,speed_ms,0,blend_radius_m)
    movel([0.063848, -1.388375, -2.540078, -0.783935, 1.570796, 1.634644],accel_mss,speed_ms,0,blend_radius_m)
    movel([0.063848, -1.409262, -2.549885, -0.753241, 1.570796, 1.634644],accel_mss,speed_ms,0,blend_radius_m)
    movel([0.063684, -1.411435, -2.548257, -0.752697, 1.570796, 1.634480],accel_mss,speed_ms,0,blend_radius_m)
    movel([0.063345, -1.412242, -2.547651, -0.752497, 1.570796, 1.634141],accel_mss,speed_ms,0,blend_radius_m)
    movel([0.063043, -1.412566, -2.547406, -0.752416, 1.570796, 1.633839],accel_mss,speed_ms,0,blend_radius_m)
    movel([0.062457, -1.412975, -2.547099, -0.752315, 1.570796, 1.633253],accel_mss,speed_ms,0,blend_radius_m)
    movel([0.061889, -1.413143, -2.546972, -0.752274, 1.570796, 1.632685],accel_mss,speed_ms,0,blend_radius_m)
    movel([0.061338, -1.413070, -2.547027, -0.752292, 1.570796, 1.632134],accel_mss,speed_ms,0,blend_radius_m)
    movel([0.061071, -1.412914, -2.547144, -0.752330, 1.570796, 1.631867],accel_mss,speed_ms,0,blend_radius_m)
    movel([0.060839, -1.412277, -2.547624, -0.752488, 1.570796, 1.631635],accel_mss,speed_ms,0,blend_radius_m)
    movel([0.060995, -1.410109, -2.549252, -0.753028, 1.570796, 1.631791],accel_mss,speed_ms,0,blend_radius_m)
    movel([0.060995, -1.389237, -2.539454, -0.783699, 1.570796, 1.631791],accel_mss,speed_ms,0,blend_radius_m)
    movel([0.060873, -1.390953, -2.538206, -0.783230, 1.570796, 1.631670],accel_mss,speed_ms,0,blend_radius_m)
    movel([0.060873, -1.411796, -2.547986, -0.752607, 1.570796, 1.631670],accel_mss,speed_ms,0,blend_radius_m)
    movel([0.057630, -1.414408, -2.546018, -0.751964, 1.570796, 1.628426],accel_mss,speed_ms,0,blend_radius_m)
    movel([0.057630, -1.393611, -2.536266, -0.782513, 1.570796, 1.628426],accel_mss,speed_ms,0,blend_radius_m)
    movel([0.063377, -1.394744, -2.535436, -0.782210, 1.570796, 1.634173],accel_mss,speed_ms,0,blend_radius_m)
    movel([0.063377, -1.415521, -2.545176, -0.751692, 1.570796, 1.634173],accel_mss,speed_ms,0,blend_radius_m)
    movel([0.063129, -1.415125, -2.545476, -0.751789, 1.570796, 1.633926],accel_mss,speed_ms,0,blend_radius_m)
    movel([0.062598, -1.414812, -2.545712, -0.751865, 1.570796, 1.633395],accel_mss,speed_ms,0,blend_radius_m)
    movel([0.062049, -1.414739, -2.545767, -0.751883, 1.570796, 1.632845],accel_mss,speed_ms,0,blend_radius_m)
    movel([0.061216, -1.414750, -2.545759, -0.751880, 1.570796, 1.632012],accel_mss,speed_ms,0,blend_radius_m)
    movel([0.059799, -1.415170, -2.545441, -0.751778, 1.570796, 1.630595],accel_mss,speed_ms,0,blend_radius_m)
    movel([0.058932, -1.415662, -2.545069, -0.751658, 1.570796, 1.629728],accel_mss,speed_ms,0,blend_radius_m)
    movel([0.058349, -1.416069, -2.544761, -0.751560, 1.570796, 1.629145],accel_mss,speed_ms,0,blend_radius_m)
    movel([0.057750, -1.416715, -2.544271, -0.751403, 1.570796, 1.628546],accel_mss,speed_ms,0,blend_radius_m)
    movel([0.057434, -1.417276, -2.543844, -0.751268, 1.570796, 1.628230],accel_mss,speed_ms,0,blend_radius_m)
    movel([0.057369, -1.418230, -2.543119, -0.751040, 1.570796, 1.628165],accel_mss,speed_ms,0,blend_radius_m)
    movel([0.057619, -1.418623, -2.542820, -0.750946, 1.570796, 1.628415],accel_mss,speed_ms,0,blend_radius_m)
    movel([0.058151, -1.418931, -2.542585, -0.750873, 1.570796, 1.628947],accel_mss,speed_ms,0,blend_radius_m)
    movel([0.058698, -1.419003, -2.542530, -0.750856, 1.570796, 1.629495],accel_mss,speed_ms,0,blend_radius_m)
    movel([0.059528, -1.418991, -2.542539, -0.750859, 1.570796, 1.630325],accel_mss,speed_ms,0,blend_radius_m)
    movel([0.060939, -1.418576, -2.542856, -0.750958, 1.570796, 1.631735],accel_mss,speed_ms,0,blend_radius_m)
    movel([0.061803, -1.418088, -2.543227, -0.751074, 1.570796, 1.632600],accel_mss,speed_ms,0,blend_radius_m)
    movel([0.062386, -1.417684, -2.543535, -0.751171, 1.570796, 1.633182],accel_mss,speed_ms,0,blend_radius_m)
    movel([0.062986, -1.417040, -2.544024, -0.751325, 1.570796, 1.633783],accel_mss,speed_ms,0,blend_radius_m)
    movel([0.063305, -1.416479, -2.544450, -0.751460, 1.570796, 1.634101],accel_mss,speed_ms,0,blend_radius_m)
    movel([0.063377, -1.415521, -2.545176, -0.751692, 1.570796, 1.634173],accel_mss,speed_ms,0,blend_radius_m)
    movel([0.063377, -1.394744, -2.535436, -0.782210, 1.570796, 1.634173],accel_mss,speed_ms,0,blend_radius_m)
    movel([0.063073, -1.398878, -2.532391, -0.781121, 1.570796, 1.633869],accel_mss,speed_ms,0,blend_radius_m)
    movel([0.063073, -1.419583, -2.542088, -0.750718, 1.570796, 1.633869],accel_mss,speed_ms,0,blend_radius_m)
    movel([0.057159, -1.421320, -2.540760, -0.750309, 1.570796, 1.627955],accel_mss,speed_ms,0,blend_radius_m)
    movel([0.057159, -1.400645, -2.531081, -0.780662, 1.570796, 1.627955],accel_mss,speed_ms,0,blend_radius_m)
    movel([0.063073, -1.398878, -2.532391, -0.781121, 1.570796, 1.633869],accel_mss,speed_ms,0,blend_radius_m)
    movel([0.063073, -1.419583, -2.542088, -0.750718, 1.570796, 1.633869],accel_mss,speed_ms,0,blend_radius_m)
    movel([0.062913, -1.421724, -2.540450, -0.750215, 1.570796, 1.633709],accel_mss,speed_ms,0,blend_radius_m)
    movel([0.062579, -1.422518, -2.539841, -0.750030, 1.570796, 1.633375],accel_mss,speed_ms,0,blend_radius_m)
    movel([0.062281, -1.422837, -2.539596, -0.749956, 1.570796, 1.633077],accel_mss,speed_ms,0,blend_radius_m)
    movel([0.061702, -1.423237, -2.539289, -0.749863, 1.570796, 1.632498],accel_mss,speed_ms,0,blend_radius_m)
    movel([0.061141, -1.423401, -2.539163, -0.749825, 1.570796, 1.631937],accel_mss,speed_ms,0,blend_radius_m)
    movel([0.060596, -1.423328, -2.539219, -0.749842, 1.570796, 1.631393],accel_mss,speed_ms,0,blend_radius_m)
    movel([0.060333, -1.423173, -2.539338, -0.749878, 1.570796, 1.631129],accel_mss,speed_ms,0,blend_radius_m)
    movel([0.060103, -1.422544, -2.539821, -0.750024, 1.570796, 1.630899],accel_mss,speed_ms,0,blend_radius_m)
    movel([0.060103, -1.401891, -2.530156, -0.780342, 1.570796, 1.630899],accel_mss,speed_ms,0,blend_radius_m)
    movel([0.060255, -1.399717, -2.531770, -0.780903, 1.570796, 1.631052],accel_mss,speed_ms,0,blend_radius_m)
    movel([0.060255, -1.420408, -2.541458, -0.750523, 1.570796, 1.631052],accel_mss,speed_ms,0,blend_radius_m)
    movel([0.060103, -1.422544, -2.539821, -0.750024, 1.570796, 1.630899],accel_mss,speed_ms,0,blend_radius_m)
    movel([0.059772, -1.423337, -2.539212, -0.749840, 1.570796, 1.630568],accel_mss,speed_ms,0,blend_radius_m)
    movel([0.059474, -1.423656, -2.538967, -0.749766, 1.570796, 1.630271],accel_mss,speed_ms,0,blend_radius_m)
    movel([0.058897, -1.424057, -2.538658, -0.749674, 1.570796, 1.629693],accel_mss,speed_ms,0,blend_radius_m)
    movel([0.058056, -1.424303, -2.538468, -0.749617, 1.570796, 1.628852],accel_mss,speed_ms,0,blend_radius_m)
    movel([0.057511, -1.424232, -2.538523, -0.749634, 1.570796, 1.628307],accel_mss,speed_ms,0,blend_radius_m)
    movel([0.057247, -1.424078, -2.538642, -0.749669, 1.570796, 1.628043],accel_mss,speed_ms,0,blend_radius_m)
    movel([0.057014, -1.423452, -2.539124, -0.749813, 1.570796, 1.627811],accel_mss,speed_ms,0,blend_radius_m)
    movel([0.057159, -1.421320, -2.540760, -0.750309, 1.570796, 1.627955],accel_mss,speed_ms,0,blend_radius_m)
    movel([0.057159, -1.400645, -2.531081, -0.780662, 1.570796, 1.627955],accel_mss,speed_ms,0,blend_radius_m)
    movel([0.062613, -1.405155, -2.527721, -0.779514, 1.570796, 1.633410],accel_mss,speed_ms,0,blend_radius_m)
    movel([0.062613, -1.425751, -2.537352, -0.749286, 1.570796, 1.633410],accel_mss,speed_ms,0,blend_radius_m)
    movel([0.062369, -1.425359, -2.537654, -0.749376, 1.570796, 1.633165],accel_mss,speed_ms,0,blend_radius_m)
    movel([0.061843, -1.425049, -2.537894, -0.749446, 1.570796, 1.632640],accel_mss,speed_ms,0,blend_radius_m)
    movel([0.061301, -1.424975, -2.537951, -0.749463, 1.570796, 1.632097],accel_mss,speed_ms,0,blend_radius_m)
    movel([0.060478, -1.424984, -2.537944, -0.749461, 1.570796, 1.631274],accel_mss,speed_ms,0,blend_radius_m)
    movel([0.059078, -1.425392, -2.537629, -0.749368, 1.570796, 1.629874],accel_mss,speed_ms,0,blend_radius_m)
    movel([0.058222, -1.425873, -2.537257, -0.749258, 1.570796, 1.629018],accel_mss,speed_ms,0,blend_radius_m)
    movel([0.057646, -1.426273, -2.536948, -0.749168, 1.570796, 1.628442],accel_mss,speed_ms,0,blend_radius_m)
    movel([0.057055, -1.426908, -2.536457, -0.749024, 1.570796, 1.627851],accel_mss,speed_ms,0,blend_radius_m)
    movel([0.056743, -1.427460, -2.536029, -0.748900, 1.570796, 1.627540],accel_mss,speed_ms,0,blend_radius_m)
    movel([0.056680, -1.428400, -2.535300, -0.748689, 1.570796, 1.627476],accel_mss,speed_ms,0,blend_radius_m)
    movel([0.056927, -1.428788, -2.534999, -0.748602, 1.570796, 1.627724],accel_mss,speed_ms,0,blend_radius_m)
    movel([0.057453, -1.429095, -2.534760, -0.748534, 1.570796, 1.628249],accel_mss,speed_ms,0,blend_radius_m)
    movel([0.057994, -1.429167, -2.534704, -0.748518, 1.570796, 1.628791],accel_mss,speed_ms,0,blend_radius_m)
    movel([0.058814, -1.429158, -2.534711, -0.748520, 1.570796, 1.629610],accel_mss,speed_ms,0,blend_radius_m)
    movel([0.060207, -1.428753, -2.535026, -0.748610, 1.570796, 1.631004],accel_mss,speed_ms,0,blend_radius_m)
    movel([0.061061, -1.428276, -2.535396, -0.748717, 1.570796, 1.631857],accel_mss,speed_ms,0,blend_radius_m)
    movel([0.061636, -1.427879, -2.535704, -0.748805, 1.570796, 1.632432],accel_mss,speed_ms,0,blend_radius_m)
    movel([0.062229, -1.427247, -2.536195, -0.748948, 1.570796, 1.633025],accel_mss,speed_ms,0,blend_radius_m)
    movel([0.062543, -1.426695, -2.536622, -0.749072, 1.570796, 1.633340],accel_mss,speed_ms,0,blend_radius_m)
    movel([0.062613, -1.425751, -2.537352, -0.749286, 1.570796, 1.633410],accel_mss,speed_ms,0,blend_radius_m)
    movel([0.062613, -1.405155, -2.527721, -0.779514, 1.570796, 1.633410],accel_mss,speed_ms,0,blend_radius_m)
    movel([0.062247, -1.410186, -2.523937, -0.778266, 1.570796, 1.633044],accel_mss,speed_ms,0,blend_radius_m)
    movel([0.062247, -1.430693, -2.533516, -0.748180, 1.570796, 1.633044],accel_mss,speed_ms,0,blend_radius_m)
    movel([0.056412, -1.432381, -2.532197, -0.747811, 1.570796, 1.627209],accel_mss,speed_ms,0,blend_radius_m)
    movel([0.056412, -1.411904, -2.522636, -0.777849, 1.570796, 1.627209],accel_mss,speed_ms,0,blend_radius_m)
    movel([0.062369, -1.408513, -2.525199, -0.778677, 1.570796, 1.633165],accel_mss,speed_ms,0,blend_radius_m)
    movel([0.062369, -1.429049, -2.534796, -0.748544, 1.570796, 1.633165],accel_mss,speed_ms,0,blend_radius_m)
    movel([0.062126, -1.432333, -2.532235, -0.747821, 1.570796, 1.632923],accel_mss,speed_ms,0,blend_radius_m)
    movel([0.062126, -1.411855, -2.522673, -0.777861, 1.570796, 1.632923],accel_mss,speed_ms,0,blend_radius_m)
    movel([0.081962, -1.182426, -2.661604, -0.868359, 1.570796, 1.652759],accel_mss,speed_ms,0,blend_radius_m)
    movel([0.081962, -1.206017, -2.673677, -0.832695, 1.570796, 1.652759],accel_mss,speed_ms,0,blend_radius_m)
    movel([0.082919, -1.205813, -2.673775, -0.832801, 1.570796, 1.653716],accel_mss,speed_ms,0,blend_radius_m)
    movel([0.083705, -1.206474, -2.673456, -0.832459, 1.570796, 1.654501],accel_mss,speed_ms,0,blend_radius_m)
    movel([0.082948, -1.214677, -2.669453, -0.828259, 1.570796, 1.653744],accel_mss,speed_ms,0,blend_radius_m)
    movel([0.081115, -1.215390, -2.669101, -0.827898, 1.570796, 1.651911],accel_mss,speed_ms,0,blend_radius_m)
    movel([0.081855, -1.207202, -2.673104, -0.832083, 1.570796, 1.652651],accel_mss,speed_ms,0,blend_radius_m)
    movel([0.074630, -1.210067, -2.671712, -0.830610, 1.570796, 1.645426],accel_mss,speed_ms,0,blend_radius_m)
    movel([0.074213, -1.215096, -2.669246, -0.828047, 1.570796, 1.645010],accel_mss,speed_ms,0,blend_radius_m)
    movel([0.080261, -1.212690, -2.670429, -0.829269, 1.570796, 1.651058],accel_mss,speed_ms,0,blend_radius_m)
    movel([0.080158, -1.213855, -2.669858, -0.828677, 1.570796, 1.650954],accel_mss,speed_ms,0,blend_radius_m)
    movel([0.074120, -1.216230, -2.668686, -0.827472, 1.570796, 1.644916],accel_mss,speed_ms,0,blend_radius_m)
    movel([0.073155, -1.216442, -2.668582, -0.827365, 1.570796, 1.643951],accel_mss,speed_ms,0,blend_radius_m)
    movel([0.072371, -1.215834, -2.668882, -0.827673, 1.570796, 1.643167],accel_mss,speed_ms,0,blend_radius_m)
    movel([0.072777, -1.210807, -2.671351, -0.830231, 1.570796, 1.643574],accel_mss,speed_ms,0,blend_radius_m)
    movel([0.073696, -1.209521, -2.671978, -0.830890, 1.570796, 1.644492],accel_mss,speed_ms,0,blend_radius_m)
    movel([0.074725, -1.208922, -2.672269, -0.831198, 1.570796, 1.645521],accel_mss,speed_ms,0,blend_radius_m)
    movel([0.073696, -1.209521, -2.671978, -0.830890, 1.570796, 1.644492],accel_mss,speed_ms,0,blend_radius_m)
    movel([0.072777, -1.210807, -2.671351, -0.830231, 1.570796, 1.643574],accel_mss,speed_ms,0,blend_radius_m)
    movel([0.072371, -1.215834, -2.668882, -0.827673, 1.570796, 1.643167],accel_mss,speed_ms,0,blend_radius_m)
    movel([0.073155, -1.216442, -2.668582, -0.827365, 1.570796, 1.643951],accel_mss,speed_ms,0,blend_radius_m)
    movel([0.074120, -1.216230, -2.668686, -0.827472, 1.570796, 1.644916],accel_mss,speed_ms,0,blend_radius_m)
    movel([0.080158, -1.213855, -2.669858, -0.828677, 1.570796, 1.650954],accel_mss,speed_ms,0,blend_radius_m)
    movel([0.080261, -1.212690, -2.670429, -0.829269, 1.570796, 1.651058],accel_mss,speed_ms,0,blend_radius_m)
    movel([0.074213, -1.215096, -2.669246, -0.828047, 1.570796, 1.645010],accel_mss,speed_ms,0,blend_radius_m)
    movel([0.074630, -1.210067, -2.671712, -0.830610, 1.570796, 1.645426],accel_mss,speed_ms,0,blend_radius_m)
    movel([0.081855, -1.207202, -2.673104, -0.832083, 1.570796, 1.652651],accel_mss,speed_ms,0,blend_radius_m)
    movel([0.081115, -1.215390, -2.669101, -0.827898, 1.570796, 1.651911],accel_mss,speed_ms,0,blend_radius_m)
    movel([0.082948, -1.214677, -2.669453, -0.828259, 1.570796, 1.653744],accel_mss,speed_ms,0,blend_radius_m)
    movel([0.083705, -1.206474, -2.673456, -0.832459, 1.570796, 1.654501],accel_mss,speed_ms,0,blend_radius_m)
    movel([0.082919, -1.205813, -2.673775, -0.832801, 1.570796, 1.653716],accel_mss,speed_ms,0,blend_radius_m)
    movel([0.081962, -1.206017, -2.673677, -0.832695, 1.570796, 1.652759],accel_mss,speed_ms,0,blend_radius_m)
    movel([0.081962, -1.182426, -2.661604, -0.868359, 1.570796, 1.652759],accel_mss,speed_ms,0,blend_radius_m)
    movel([0.074699, -1.185364, -2.660224, -0.866801, 1.570796, 1.645496],accel_mss,speed_ms,0,blend_radius_m)
    movel([0.074699, -1.208933, -2.672264, -0.831192, 1.570796, 1.645496],accel_mss,speed_ms,0,blend_radius_m)
    movel([0.081962, -1.206017, -2.673677, -0.832695, 1.570796, 1.652759],accel_mss,speed_ms,0,blend_radius_m)
    movel([0.074699, -1.208933, -2.672264, -0.831192, 1.570796, 1.645496],accel_mss,speed_ms,0,blend_radius_m)
    movel([0.081962, -1.206017, -2.673677, -0.832695, 1.570796, 1.652759],accel_mss,speed_ms,0,blend_radius_m)
    movel([0.074699, -1.208933, -2.672264, -0.831192, 1.570796, 1.645496],accel_mss,speed_ms,0,blend_radius_m)
    movel([0.074699, -1.185364, -2.660224, -0.866801, 1.570796, 1.645496],accel_mss,speed_ms,0,blend_radius_m)
    movel([0.086559, -1.180588, -2.662463, -0.869339, 1.570796, 1.657355],accel_mss,speed_ms,0,blend_radius_m)
